KUKA KRL program: f1_Kuka_APT206T03S06.SRC

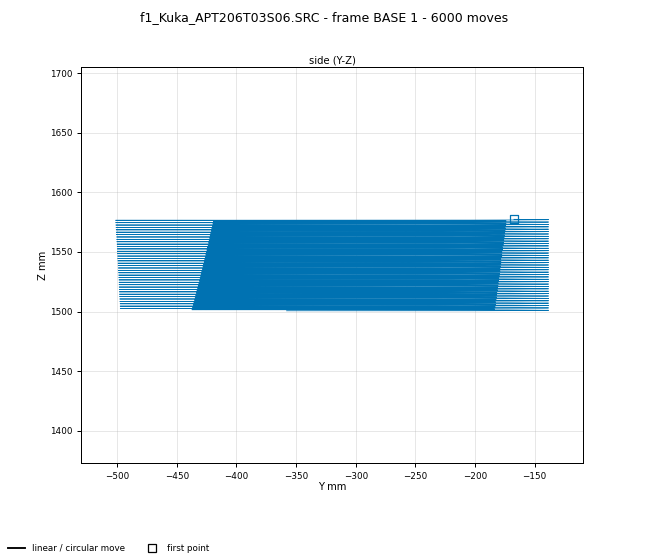
[picture p0: tool path of f1_Kuka_APT206T03S06.SRC in frame BASE 1, 6000 of 6001 moves have a stored position in this frame; points joined in program order, loops and branches not executed]
&ACCESS RVP
&REL 2
&PARAM TEMPLATE = C:\KRC\Roboter\Template\vorgabe
&PARAM EDITMASK = *
DEF f1_Kuka_APT206T03S06()


;FOLD INI;%{PE}%V3.2.0,%MKUKATPBASIS,%CINIT,%VCOMMON,%P
  ;FOLD BAS INI;%{E}%V3.2.0,%MKUKATPBASIS,%CINIT,%VINIT,%P
    GLOBAL INTERRUPT DECL 3 WHEN $STOPMESS==TRUE DO IR_STOPM ( )
    INTERRUPT ON 3
    BAS (#INITMOV,0 )
  ;ENDFOLD (BAS INI)
  ;FOLD USER INI;%{E}%V3.2.0,%MKUKATPUSER,%CINIT,%VINIT,%P
    ;Make your modifications here
  ;ENDFOLD (USER INI)
;ENDFOLD (INI)


;*** Make Null PTP Move
  PTP $pos_act

;*** Auto Load The Correct TOOL Data
  $tool=tool_data[3]

;*** Auto Load The Correct BASE Data
  $base=base_data[1]

  $ADVANCE = 5

;*** Restate Last Velocity
MMPM(30000.0)
SetRPM(6000)
LIN {X 0.095,Y -167.291,Z 1577.353,A 0.000,B 0.000,C 90.000,E1 243.512} C_DIS
LIN {X 0.027,Y -166.668,Z 1577.348,A 0.000,B 0.000,C 90.000,E1 242.666} C_DIS
LIN {X -0.056,Y -162.651,Z 1577.324,A 0.000,B 0.000,C 90.000,E1 238.329} C_DIS
LIN {X 0.006,Y -161.340,Z 1577.314,A 0.000,B 0.000,C 90.000,E1 236.548} C_DIS
LIN {X 0.048,Y -157.334,Z 1577.290,A 0.000,B 0.000,C 90.000,E1 232.110} C_DIS
LIN {X -0.019,Y -155.318,Z 1577.275,A 0.000,B 0.000,C 90.000,E1 229.461} C_DIS
LIN {X 0.019,Y -151.672,Z 1577.250,A 0.000,B 0.000,C 90.000,E1 224.960} C_DIS
LIN {X -0.040,Y -150.538,Z 1577.240,A 0.000,B 0.000,C 90.000,E1 223.176} C_DIS
LIN {X -0.007,Y -147.263,Z 1577.215,A 0.000,B 0.000,C 90.000,E1 218.624} C_DIS
LIN {X 0.050,Y -145.289,Z 1577.194,A 0.000,B 0.000,C 90.000,E1 214.945} C_DIS
LIN {X -0.041,Y -142.389,Z 1577.164,A 0.000,B 0.000,C 90.000,E1 209.461} C_DIS
LIN {X 0.005,Y -141.367,Z 1577.148,A 0.000,B 0.000,C 90.000,E1 206.668} C_DIS
LIN {X -0.017,Y -139.344,Z 1577.112,A 0.000,B 0.000,C 90.000,E1 200.174} C_DIS
LIN {X -0.011,Y -139.015,Z 1577.102,A 0.000,B 0.000,C 90.000,E1 198.308} C_DIS
LIN {X -0.015,Y -138.342,Z 1577.055,A 0.000,B 0.000,C 90.000,E1 189.905} C_DIS
LIN {X 0.004,Y -139.395,Z 1577.008,A 0.000,B 0.000,C 90.000,E1 181.489} C_DIS
LIN {X 0.058,Y -141.296,Z 1576.972,A 0.000,B 0.000,C 90.000,E1 174.951} C_DIS
LIN {X 0.016,Y -142.659,Z 1576.957,A 0.000,B 0.000,C 90.000,E1 172.186} C_DIS
LIN {X -0.034,Y -145.001,Z 1576.931,A 0.000,B 0.000,C 90.000,E1 167.589} C_DIS
LIN {X -0.045,Y -147.628,Z 1576.911,A 0.000,B 0.000,C 90.000,E1 163.921} C_DIS
LIN {X 0.033,Y -150.257,Z 1576.890,A 0.000,B 0.000,C 90.000,E1 160.242} C_DIS
LIN {X 0.047,Y -153.653,Z 1576.870,A 0.000,B 0.000,C 90.000,E1 156.613} C_DIS
LIN {X -0.036,Y -157.069,Z 1576.850,A 0.000,B 0.000,C 90.000,E1 153.050} C_DIS
LIN {X 0.042,Y -161.201,Z 1576.830,A 0.000,B 0.000,C 90.000,E1 149.459} C_DIS
LIN {X -0.009,Y -163.293,Z 1576.821,A 0.000,B 0.000,C 90.000,E1 147.709} C_DIS
LIN {X 0.001,Y -167.738,Z 1576.801,A 0.000,B 0.000,C 90.000,E1 144.196} C_DIS
LIN {X -0.087,Y -171.556,Z 1576.787,A 0.000,B 0.000,C 90.000,E1 141.618} C_DIS
LIN {X -0.046,Y -176.501,Z 1576.767,A 0.000,B 0.000,C 90.000,E1 138.162} C_DIS
LIN {X 0.080,Y -180.798,Z 1576.753,A 0.000,B 0.000,C 90.000,E1 135.567} C_DIS
LIN {X 0.065,Y -186.206,Z 1576.735,A 0.000,B 0.000,C 90.000,E1 132.204} C_DIS
LIN {X 0.004,Y -190.844,Z 1576.721,A 0.000,B 0.000,C 90.000,E1 129.725} C_DIS
LIN {X 0.038,Y -196.604,Z 1576.702,A 0.000,B 0.000,C 90.000,E1 126.423} C_DIS
LIN {X 0.006,Y -201.369,Z 1576.689,A 0.000,B 0.000,C 90.000,E1 123.992} C_DIS
LIN {X 0.013,Y -204.164,Z 1576.680,A 0.000,B 0.000,C 90.000,E1 122.418} C_DIS
LIN {X -0.014,Y -320.855,Z 1576.680,A 0.000,B 0.000,C 90.000,E1 122.418} C_DIS
LIN {X -0.039,Y -323.066,Z 1576.680,A 0.000,B 0.000,C 90.000,E1 122.388} C_DIS
LIN {X 0.035,Y -325.993,Z 1576.679,A 0.000,B 0.000,C 90.000,E1 122.260} C_DIS
LIN {X 0.100,Y -329.452,Z 1576.678,A 0.000,B 0.000,C 90.000,E1 122.005} C_DIS
LIN {X 0.070,Y -333.103,Z 1576.676,A 0.000,B 0.000,C 90.000,E1 121.592} C_DIS
LIN {X -0.223,Y -334.975,Z 1576.674,A 0.000,B 0.000,C 90.000,E1 121.337} C_DIS
LIN {X -0.056,Y -336.437,Z 1576.672,A 0.000,B 0.000,C 90.000,E1 121.003} C_DIS
LIN {X 0.068,Y -349.361,Z 1576.655,A 0.000,B 0.000,C 90.000,E1 117.897} C_DIS
LIN {X -0.105,Y -362.479,Z 1576.640,A 0.000,B 0.000,C 90.000,E1 115.207} C_DIS
LIN {X 0.113,Y -377.146,Z 1576.625,A 0.000,B 0.000,C 90.000,E1 112.514} C_DIS
LIN {X -0.183,Y -391.580,Z 1576.612,A 0.000,B 0.000,C 90.000,E1 110.248} C_DIS
LIN {X 0.123,Y -407.435,Z 1576.600,A 0.000,B 0.000,C 90.000,E1 107.946} C_DIS
LIN {X -0.208,Y -424.819,Z 1576.588,A 0.000,B 0.000,C 90.000,E1 105.788} C_DIS
LIN {X 0.185,Y -443.846,Z 1576.576,A 0.000,B 0.000,C 90.000,E1 103.592} C_DIS
LIN {X 0.113,Y -463.869,Z 1576.564,A 0.000,B 0.000,C 90.000,E1 101.591} C_DIS
LIN {X -0.162,Y -487.025,Z 1576.553,A 0.000,B 0.000,C 90.000,E1 99.557} C_DIS
LIN {X -0.235,Y -494.749,Z 1576.549,A 0.000,B 0.000,C 90.000,E1 98.916} C_DIS
LIN {X -0.117,Y -496.703,Z 1576.548,A 0.000,B 0.000,C 90.000,E1 98.681} C_DIS
LIN {X -0.073,Y -498.197,Z 1576.547,A 0.000,B 0.000,C 90.000,E1 98.454} C_DIS
LIN {X -0.153,Y -499.446,Z 1576.546,A 0.000,B 0.000,C 90.000,E1 98.219} C_DIS
LIN {X 0.192,Y -500.355,Z 1576.544,A 0.000,B 0.000,C 90.000,E1 97.936} C_DIS
LIN {X 0.043,Y -501.319,Z 1576.542,A 0.000,B 0.000,C 90.000,E1 97.466} C_DIS
LIN {X -0.168,Y -501.267,Z 1576.539,A 0.000,B 0.000,C 90.000,E1 97.004} C_DIS
LIN {X 0.122,Y -500.195,Z 1576.536,A 0.000,B 0.000,C 90.000,E1 96.486} C_DIS
LIN {X -0.009,Y -499.226,Z 1576.535,A 0.000,B 0.000,C 90.000,E1 96.258} C_DIS
LIN {X -0.137,Y -497.907,Z 1576.533,A 0.000,B 0.000,C 90.000,E1 96.030} C_DIS
LIN {X 0.044,Y -481.661,Z 1576.520,A 0.000,B 0.000,C 90.000,E1 93.555} C_DIS
LIN {X -0.017,Y -471.774,Z 1576.511,A 0.000,B 0.000,C 90.000,E1 92.064} C_DIS
LIN {X -0.040,Y -463.226,Z 1576.504,A 0.000,B 0.000,C 90.000,E1 90.802} C_DIS
LIN {X -0.187,Y -454.292,Z 1576.497,A 0.000,B 0.000,C 90.000,E1 89.542} C_DIS
LIN {X -0.018,Y -444.960,Z 1576.490,A 0.000,B 0.000,C 90.000,E1 88.224} C_DIS
LIN {X 0.026,Y -435.162,Z 1576.483,A 0.000,B 0.000,C 90.000,E1 86.906} C_DIS
LIN {X -0.192,Y -421.167,Z 1576.472,A 0.000,B 0.000,C 90.000,E1 85.065} C_DIS
LIN {X 0.006,Y -401.901,Z 1576.457,A 0.000,B 0.000,C 90.000,E1 82.299} C_DIS
LIN {X 0.185,Y -383.905,Z 1576.442,A 0.000,B 0.000,C 90.000,E1 79.454} C_DIS
LIN {X -0.013,Y -368.716,Z 1576.427,A 0.000,B 0.000,C 90.000,E1 76.881} C_DIS
LIN {X -0.045,Y -355.690,Z 1576.414,A 0.000,B 0.000,C 90.000,E1 74.519} C_DIS
LIN {X -0.198,Y -342.958,Z 1576.401,A 0.000,B 0.000,C 90.000,E1 72.127} C_DIS
LIN {X -0.144,Y -329.138,Z 1576.385,A 0.000,B 0.000,C 90.000,E1 69.337} C_DIS
LIN {X -0.054,Y -317.496,Z 1576.371,A 0.000,B 0.000,C 90.000,E1 66.794} C_DIS
LIN {X 0.006,Y -306.059,Z 1576.357,A 0.000,B 0.000,C 90.000,E1 64.204} C_DIS
LIN {X 0.045,Y -296.354,Z 1576.344,A 0.000,B 0.000,C 90.000,E1 61.897} C_DIS
LIN {X 0.140,Y -286.545,Z 1576.331,A 0.000,B 0.000,C 90.000,E1 59.537} C_DIS
LIN {X 0.017,Y -275.221,Z 1576.316,A 0.000,B 0.000,C 90.000,E1 56.834} C_DIS
LIN {X -0.067,Y -266.836,Z 1576.304,A 0.000,B 0.000,C 90.000,E1 54.769} C_DIS
LIN {X 0.128,Y -254.472,Z 1576.286,A 0.000,B 0.000,C 90.000,E1 51.537} C_DIS
LIN {X -0.100,Y -242.916,Z 1576.268,A 0.000,B 0.000,C 90.000,E1 48.324} C_DIS
LIN {X 0.003,Y -232.326,Z 1576.250,A 0.000,B 0.000,C 90.000,E1 44.960} C_DIS
LIN {X 0.061,Y -223.742,Z 1576.233,A 0.000,B 0.000,C 90.000,E1 41.919} C_DIS
LIN {X 0.110,Y -215.941,Z 1576.216,A 0.000,B 0.000,C 90.000,E1 38.830} C_DIS
LIN {X 0.031,Y -208.847,Z 1576.198,A 0.000,B 0.000,C 90.000,E1 35.724} C_DIS
LIN {X 0.045,Y -202.542,Z 1576.181,A 0.000,B 0.000,C 90.000,E1 32.546} C_DIS
LIN {X 0.031,Y -197.052,Z 1576.163,A 0.000,B 0.000,C 90.000,E1 29.333} C_DIS
LIN {X -0.059,Y -192.330,Z 1576.145,A 0.000,B 0.000,C 90.000,E1 26.104} C_DIS
LIN {X -0.007,Y -187.330,Z 1576.122,A 0.000,B 0.000,C 90.000,E1 21.972} C_DIS
LIN {X -0.033,Y -183.183,Z 1576.099,A 0.000,B 0.000,C 90.000,E1 17.819} C_DIS
LIN {X 0.054,Y -179.813,Z 1576.076,A 0.000,B 0.000,C 90.000,E1 13.592} C_DIS
LIN {X -0.068,Y -176.374,Z 1576.043,A 0.000,B 0.000,C 90.000,E1 7.701} C_DIS
LIN {X -0.029,Y -173.971,Z 1576.005,A 0.000,B 0.000,C 90.000,E1 0.859} C_DIS
LIN {X 0.097,Y -175.150,Z 1575.940,A 0.000,B 0.000,C 90.000,E1 349.218} C_DIS
LIN {X -0.078,Y -177.819,Z 1575.912,A 0.000,B 0.000,C 90.000,E1 344.157} C_DIS
LIN {X 0.041,Y -181.126,Z 1575.888,A 0.000,B 0.000,C 90.000,E1 339.880} C_DIS
LIN {X 0.075,Y -185.579,Z 1575.865,A 0.000,B 0.000,C 90.000,E1 335.665} C_DIS
LIN {X -0.008,Y -189.856,Z 1575.846,A 0.000,B 0.000,C 90.000,E1 332.359} C_DIS
LIN {X -0.062,Y -194.857,Z 1575.828,A 0.000,B 0.000,C 90.000,E1 329.076} C_DIS
LIN {X -0.022,Y -200.563,Z 1575.810,A 0.000,B 0.000,C 90.000,E1 325.801} C_DIS
LIN {X 0.064,Y -207.089,Z 1575.792,A 0.000,B 0.000,C 90.000,E1 322.557} C_DIS
LIN {X 0.077,Y -214.524,Z 1575.774,A 0.000,B 0.000,C 90.000,E1 319.380} C_DIS
LIN {X 0.023,Y -223.764,Z 1575.755,A 0.000,B 0.000,C 90.000,E1 315.891} C_DIS
LIN {X -0.040,Y -232.902,Z 1575.738,A 0.000,B 0.000,C 90.000,E1 312.852} C_DIS
LIN {X 0.002,Y -241.786,Z 1575.723,A 0.000,B 0.000,C 90.000,E1 310.216} C_DIS
LIN {X -0.050,Y -247.598,Z 1575.715,A 0.000,B 0.000,C 90.000,E1 308.749} C_DIS
LIN {X -0.028,Y -254.145,Z 1575.707,A 0.000,B 0.000,C 90.000,E1 307.282} C_DIS
LIN {X -0.028,Y -267.375,Z 1575.693,A 0.000,B 0.000,C 90.000,E1 304.771} C_DIS
LIN {X -0.044,Y -280.267,Z 1575.682,A 0.000,B 0.000,C 90.000,E1 302.673} C_DIS
LIN {X 0.109,Y -299.411,Z 1575.666,A 0.000,B 0.000,C 90.000,E1 299.922} C_DIS
LIN {X 0.048,Y -311.876,Z 1575.657,A 0.000,B 0.000,C 90.000,E1 298.281} C_DIS
LIN {X -0.027,Y -326.927,Z 1575.646,A 0.000,B 0.000,C 90.000,E1 296.360} C_DIS
LIN {X 0.062,Y -339.369,Z 1575.638,A 0.000,B 0.000,C 90.000,E1 294.771} C_DIS
LIN {X -0.090,Y -361.712,Z 1575.623,A 0.000,B 0.000,C 90.000,E1 292.078} C_DIS
LIN {X 0.149,Y -374.611,Z 1575.614,A 0.000,B 0.000,C 90.000,E1 290.556} C_DIS
LIN {X 0.113,Y -384.575,Z 1575.608,A 0.000,B 0.000,C 90.000,E1 289.396} C_DIS
LIN {X 0.036,Y -391.545,Z 1575.603,A 0.000,B 0.000,C 90.000,E1 288.544} C_DIS
LIN {X 0.079,Y -399.857,Z 1575.597,A 0.000,B 0.000,C 90.000,E1 287.402} C_DIS
LIN {X -0.055,Y -403.577,Z 1575.594,A 0.000,B 0.000,C 90.000,E1 286.858} C_DIS
LIN {X -0.075,Y -408.391,Z 1575.589,A 0.000,B 0.000,C 90.000,E1 286.024} C_DIS
LIN {X -0.160,Y -411.130,Z 1575.586,A 0.000,B 0.000,C 90.000,E1 285.481} C_DIS
LIN {X 0.060,Y -413.511,Z 1575.583,A 0.000,B 0.000,C 90.000,E1 284.898} C_DIS
LIN {X 0.129,Y -416.344,Z 1575.578,A 0.000,B 0.000,C 90.000,E1 284.064} C_DIS
LIN {X -0.018,Y -417.781,Z 1575.575,A 0.000,B 0.000,C 90.000,E1 283.536} C_DIS
LIN {X -0.153,Y -418.766,Z 1575.572,A 0.000,B 0.000,C 90.000,E1 283.008} C_DIS
LIN {X 0.220,Y -419.304,Z 1575.569,A 0.000,B 0.000,C 90.000,E1 282.411} C_DIS
LIN {X 0.097,Y -419.380,Z 1575.566,A 0.000,B 0.000,C 90.000,E1 281.883} C_DIS
LIN {X -0.107,Y -418.925,Z 1575.563,A 0.000,B 0.000,C 90.000,E1 281.366} C_DIS
LIN {X -0.225,Y -417.916,Z 1575.560,A 0.000,B 0.000,C 90.000,E1 280.838} C_DIS
LIN {X 0.063,Y -416.325,Z 1575.557,A 0.000,B 0.000,C 90.000,E1 280.254} C_DIS
LIN {X -0.067,Y -414.093,Z 1575.554,A 0.000,B 0.000,C 90.000,E1 279.726} C_DIS
LIN {X -0.005,Y -412.764,Z 1575.552,A 0.000,B 0.000,C 90.000,E1 279.443} C_DIS
LIN {X -0.157,Y -409.484,Z 1575.549,A 0.000,B 0.000,C 90.000,E1 278.916} C_DIS
LIN {X 0.014,Y -405.457,Z 1575.546,A 0.000,B 0.000,C 90.000,E1 278.341} C_DIS
LIN {X -0.179,Y -400.748,Z 1575.543,A 0.000,B 0.000,C 90.000,E1 277.814} C_DIS
LIN {X 0.036,Y -395.299,Z 1575.540,A 0.000,B 0.000,C 90.000,E1 277.239} C_DIS
LIN {X 0.065,Y -389.417,Z 1575.537,A 0.000,B 0.000,C 90.000,E1 276.720} C_DIS
LIN {X -0.010,Y -383.356,Z 1575.535,A 0.000,B 0.000,C 90.000,E1 276.258} C_DIS
LIN {X -0.011,Y -373.859,Z 1575.531,A 0.000,B 0.000,C 90.000,E1 275.625} C_DIS
LIN {X -0.175,Y -364.295,Z 1575.528,A 0.000,B 0.000,C 90.000,E1 275.106} C_DIS
LIN {X 0.037,Y -354.579,Z 1575.526,A 0.000,B 0.000,C 90.000,E1 274.588} C_DIS
LIN {X -0.165,Y -345.037,Z 1575.523,A 0.000,B 0.000,C 90.000,E1 274.188} C_DIS
LIN {X 0.165,Y -335.255,Z 1575.521,A 0.000,B 0.000,C 90.000,E1 273.726} C_DIS
LIN {X -0.025,Y -322.280,Z 1575.518,A 0.000,B 0.000,C 90.000,E1 273.269} C_DIS
LIN {X 0.106,Y -312.075,Z 1575.516,A 0.000,B 0.000,C 90.000,E1 272.922} C_DIS
LIN {X 0.125,Y -301.579,Z 1575.515,A 0.000,B 0.000,C 90.000,E1 272.636} C_DIS
LIN {X 0.116,Y -290.375,Z 1575.514,A 0.000,B 0.000,C 90.000,E1 272.407} C_DIS
LIN {X 0.057,Y -277.059,Z 1575.512,A 0.000,B 0.000,C 90.000,E1 272.236} C_DIS
LIN {X -0.089,Y -257.665,Z 1575.511,A 0.000,B 0.000,C 90.000,E1 272.064} C_DIS
LIN {X 0.109,Y -244.909,Z 1575.511,A 0.000,B 0.000,C 90.000,E1 271.949} C_DIS
LIN {X 0.058,Y -238.715,Z 1575.511,A 0.000,B 0.000,C 90.000,E1 271.949} C_DIS
LIN {X 0.026,Y -181.269,Z 1575.511,A 0.000,B 0.000,C 90.000,E1 271.949} C_DIS
LIN {X -0.068,Y -181.572,Z 1575.502,A 0.000,B 0.000,C 90.000,E1 270.458} C_DIS
LIN {X 0.015,Y -180.953,Z 1575.481,A 0.000,B 0.000,C 90.000,E1 266.560} C_DIS
LIN {X -0.048,Y -180.830,Z 1575.472,A 0.000,B 0.000,C 90.000,E1 264.894} C_DIS
LIN {X 0.032,Y -178.936,Z 1575.443,A 0.000,B 0.000,C 90.000,E1 259.803} C_DIS
LIN {X -0.100,Y -175.984,Z 1575.415,A 0.000,B 0.000,C 90.000,E1 254.755} C_DIS
LIN {X 0.015,Y -175.481,Z 1575.410,A 0.000,B 0.000,C 90.000,E1 253.866} C_DIS
LIN {X 0.072,Y -172.227,Z 1575.387,A 0.000,B 0.000,C 90.000,E1 249.571} C_DIS
LIN {X 0.049,Y -171.704,Z 1575.382,A 0.000,B 0.000,C 90.000,E1 248.720} C_DIS
LIN {X -0.026,Y -167.298,Z 1575.353,A 0.000,B 0.000,C 90.000,E1 243.563} C_DIS
LIN {X 0.056,Y -166.676,Z 1575.348,A 0.000,B 0.000,C 90.000,E1 242.666} C_DIS
LIN {X -0.029,Y -162.658,Z 1575.324,A 0.000,B 0.000,C 90.000,E1 238.329} C_DIS
LIN {X 0.033,Y -161.347,Z 1575.314,A 0.000,B 0.000,C 90.000,E1 236.548} C_DIS
LIN {X 0.075,Y -157.342,Z 1575.290,A 0.000,B 0.000,C 90.000,E1 232.110} C_DIS
LIN {X 0.008,Y -155.327,Z 1575.275,A 0.000,B 0.000,C 90.000,E1 229.461} C_DIS
LIN {X -0.062,Y -151.679,Z 1575.250,A 0.000,B 0.000,C 90.000,E1 225.000} C_DIS
LIN {X -0.014,Y -150.543,Z 1575.240,A 0.000,B 0.000,C 90.000,E1 223.176} C_DIS
LIN {X 0.020,Y -147.269,Z 1575.215,A 0.000,B 0.000,C 90.000,E1 218.624} C_DIS
LIN {X -0.008,Y -145.296,Z 1575.194,A 0.000,B 0.000,C 90.000,E1 214.978} C_DIS
LIN {X -0.015,Y -142.392,Z 1575.164,A 0.000,B 0.000,C 90.000,E1 209.461} C_DIS
LIN {X 0.031,Y -141.372,Z 1575.148,A 0.000,B 0.000,C 90.000,E1 206.668} C_DIS
LIN {X 0.009,Y -139.346,Z 1575.112,A 0.000,B 0.000,C 90.000,E1 200.174} C_DIS
LIN {X 0.014,Y -139.018,Z 1575.102,A 0.000,B 0.000,C 90.000,E1 198.308} C_DIS
LIN {X 0.010,Y -138.343,Z 1575.055,A 0.000,B 0.000,C 90.000,E1 189.905} C_DIS
LIN {X 0.029,Y -139.392,Z 1575.008,A 0.000,B 0.000,C 90.000,E1 181.489} C_DIS
LIN {X -0.057,Y -141.291,Z 1574.972,A 0.000,B 0.000,C 90.000,E1 175.008} C_DIS
LIN {X 0.042,Y -142.654,Z 1574.957,A 0.000,B 0.000,C 90.000,E1 172.186} C_DIS
LIN {X -0.008,Y -144.994,Z 1574.931,A 0.000,B 0.000,C 90.000,E1 167.589} C_DIS
LIN {X -0.019,Y -147.621,Z 1574.911,A 0.000,B 0.000,C 90.000,E1 163.921} C_DIS
LIN {X 0.059,Y -150.248,Z 1574.890,A 0.000,B 0.000,C 90.000,E1 160.242} C_DIS
LIN {X -0.067,Y -153.643,Z 1574.870,A 0.000,B 0.000,C 90.000,E1 156.666} C_DIS
LIN {X -0.009,Y -157.059,Z 1574.850,A 0.000,B 0.000,C 90.000,E1 153.050} C_DIS
LIN {X 0.071,Y -161.189,Z 1574.830,A 0.000,B 0.000,C 90.000,E1 149.459} C_DIS
LIN {X 0.019,Y -163.281,Z 1574.821,A 0.000,B 0.000,C 90.000,E1 147.709} C_DIS
LIN {X 0.029,Y -167.725,Z 1574.801,A 0.000,B 0.000,C 90.000,E1 144.196} C_DIS
LIN {X -0.058,Y -171.543,Z 1574.787,A 0.000,B 0.000,C 90.000,E1 141.618} C_DIS
LIN {X -0.016,Y -176.486,Z 1574.768,A 0.000,B 0.000,C 90.000,E1 138.162} C_DIS
LIN {X 0.109,Y -180.783,Z 1574.753,A 0.000,B 0.000,C 90.000,E1 135.567} C_DIS
LIN {X -0.030,Y -186.190,Z 1574.735,A 0.000,B 0.000,C 90.000,E1 132.243} C_DIS
LIN {X 0.035,Y -190.827,Z 1574.721,A 0.000,B 0.000,C 90.000,E1 129.725} C_DIS
LIN {X -0.047,Y -196.587,Z 1574.703,A 0.000,B 0.000,C 90.000,E1 126.457} C_DIS
LIN {X 0.037,Y -201.354,Z 1574.689,A 0.000,B 0.000,C 90.000,E1 123.992} C_DIS
LIN {X -0.027,Y -204.096,Z 1574.680,A 0.000,B 0.000,C 90.000,E1 122.467} C_DIS
LIN {X -0.078,Y -320.847,Z 1574.680,A 0.000,B 0.000,C 90.000,E1 122.467} C_DIS
LIN {X -0.162,Y -323.865,Z 1574.680,A 0.000,B 0.000,C 90.000,E1 122.418} C_DIS
LIN {X -0.054,Y -326.764,Z 1574.679,A 0.000,B 0.000,C 90.000,E1 122.260} C_DIS
LIN {X -0.011,Y -330.385,Z 1574.677,A 0.000,B 0.000,C 90.000,E1 121.957} C_DIS
LIN {X 0.095,Y -333.985,Z 1574.675,A 0.000,B 0.000,C 90.000,E1 121.465} C_DIS
LIN {X -0.073,Y -335.662,Z 1574.673,A 0.000,B 0.000,C 90.000,E1 121.180} C_DIS
LIN {X 0.015,Y -349.958,Z 1574.654,A 0.000,B 0.000,C 90.000,E1 117.769} C_DIS
LIN {X -0.143,Y -363.150,Z 1574.639,A 0.000,B 0.000,C 90.000,E1 115.079} C_DIS
LIN {X 0.092,Y -377.897,Z 1574.624,A 0.000,B 0.000,C 90.000,E1 112.386} C_DIS
LIN {X -0.189,Y -392.407,Z 1574.612,A 0.000,B 0.000,C 90.000,E1 110.120} C_DIS
LIN {X 0.133,Y -408.345,Z 1574.599,A 0.000,B 0.000,C 90.000,E1 107.819} C_DIS
LIN {X -0.181,Y -425.818,Z 1574.587,A 0.000,B 0.000,C 90.000,E1 105.662} C_DIS
LIN {X 0.139,Y -444.926,Z 1574.575,A 0.000,B 0.000,C 90.000,E1 103.480} C_DIS
LIN {X 0.149,Y -464.980,Z 1574.564,A 0.000,B 0.000,C 90.000,E1 101.478} C_DIS
LIN {X -0.038,Y -488.170,Z 1574.552,A 0.000,B 0.000,C 90.000,E1 99.443} C_DIS
LIN {X -0.190,Y -493.404,Z 1574.550,A 0.000,B 0.000,C 90.000,E1 99.029} C_DIS
LIN {X -0.082,Y -495.600,Z 1574.549,A 0.000,B 0.000,C 90.000,E1 98.803} C_DIS
LIN {X -0.110,Y -497.434,Z 1574.547,A 0.000,B 0.000,C 90.000,E1 98.568} C_DIS
LIN {X -0.213,Y -498.815,Z 1574.546,A 0.000,B 0.000,C 90.000,E1 98.341} C_DIS
LIN {X 0.126,Y -500.604,Z 1574.543,A 0.000,B 0.000,C 90.000,E1 97.814} C_DIS
LIN {X -0.095,Y -501.274,Z 1574.541,A 0.000,B 0.000,C 90.000,E1 97.352} C_DIS
LIN {X 0.193,Y -500.943,Z 1574.538,A 0.000,B 0.000,C 90.000,E1 96.834} C_DIS
LIN {X -0.012,Y -499.559,Z 1574.535,A 0.000,B 0.000,C 90.000,E1 96.372} C_DIS
LIN {X -0.142,Y -498.401,Z 1574.534,A 0.000,B 0.000,C 90.000,E1 96.144} C_DIS
LIN {X -0.151,Y -485.465,Z 1574.523,A 0.000,B 0.000,C 90.000,E1 94.188} C_DIS
LIN {X -0.118,Y -475.726,Z 1574.515,A 0.000,B 0.000,C 90.000,E1 92.694} C_DIS
LIN {X 0.187,Y -465.673,Z 1574.506,A 0.000,B 0.000,C 90.000,E1 91.146} C_DIS
LIN {X 0.069,Y -456.832,Z 1574.499,A 0.000,B 0.000,C 90.000,E1 89.885} C_DIS
LIN {X -0.175,Y -447.619,Z 1574.492,A 0.000,B 0.000,C 90.000,E1 88.625} C_DIS
LIN {X -0.087,Y -437.962,Z 1574.485,A 0.000,B 0.000,C 90.000,E1 87.306} C_DIS
LIN {X 0.022,Y -425.988,Z 1574.476,A 0.000,B 0.000,C 90.000,E1 85.698} C_DIS
LIN {X -0.168,Y -408.379,Z 1574.463,A 0.000,B 0.000,C 90.000,E1 83.280} C_DIS
LIN {X 0.151,Y -389.972,Z 1574.447,A 0.000,B 0.000,C 90.000,E1 80.443} C_DIS
LIN {X 0.128,Y -369.444,Z 1574.428,A 0.000,B 0.000,C 90.000,E1 76.992} C_DIS
LIN {X 0.115,Y -356.384,Z 1574.415,A 0.000,B 0.000,C 90.000,E1 74.629} C_DIS
LIN {X -0.034,Y -345.224,Z 1574.403,A 0.000,B 0.000,C 90.000,E1 72.543} C_DIS
LIN {X 0.060,Y -329.742,Z 1574.386,A 0.000,B 0.000,C 90.000,E1 69.444} C_DIS
LIN {X -0.018,Y -316.635,Z 1574.370,A 0.000,B 0.000,C 90.000,E1 66.613} C_DIS
LIN {X 0.015,Y -305.186,Z 1574.356,A 0.000,B 0.000,C 90.000,E1 64.024} C_DIS
LIN {X 0.030,Y -295.451,Z 1574.343,A 0.000,B 0.000,C 90.000,E1 61.719} C_DIS
LIN {X -0.149,Y -285.589,Z 1574.330,A 0.000,B 0.000,C 90.000,E1 59.410} C_DIS
LIN {X 0.095,Y -274.341,Z 1574.315,A 0.000,B 0.000,C 90.000,E1 56.628} C_DIS
LIN {X -0.007,Y -266.015,Z 1574.303,A 0.000,B 0.000,C 90.000,E1 54.562} C_DIS
LIN {X -0.039,Y -253.733,Z 1574.285,A 0.000,B 0.000,C 90.000,E1 51.376} C_DIS
LIN {X 0.067,Y -242.256,Z 1574.267,A 0.000,B 0.000,C 90.000,E1 48.081} C_DIS
LIN {X -0.017,Y -231.760,Z 1574.249,A 0.000,B 0.000,C 90.000,E1 44.757} C_DIS
LIN {X -0.130,Y -223.234,Z 1574.232,A 0.000,B 0.000,C 90.000,E1 41.757} C_DIS
LIN {X 0.078,Y -215.496,Z 1574.215,A 0.000,B 0.000,C 90.000,E1 38.624} C_DIS
LIN {X -0.009,Y -208.484,Z 1574.197,A 0.000,B 0.000,C 90.000,E1 35.518} C_DIS
LIN {X -0.001,Y -202.268,Z 1574.180,A 0.000,B 0.000,C 90.000,E1 32.339} C_DIS
LIN {X -0.023,Y -196.843,Z 1574.162,A 0.000,B 0.000,C 90.000,E1 29.127} C_DIS
LIN {X 0.052,Y -192.183,Z 1574.144,A 0.000,B 0.000,C 90.000,E1 25.848} C_DIS
LIN {X 0.095,Y -187.263,Z 1574.121,A 0.000,B 0.000,C 90.000,E1 21.716} C_DIS
LIN {X 0.001,Y -183.167,Z 1574.098,A 0.000,B 0.000,C 90.000,E1 17.583} C_DIS
LIN {X 0.016,Y -179.309,Z 1574.070,A 0.000,B 0.000,C 90.000,E1 12.535} C_DIS
LIN {X -0.007,Y -176.097,Z 1574.037,A 0.000,B 0.000,C 90.000,E1 6.606} C_DIS
LIN {X -0.032,Y -174.013,Z 1573.997,A 0.000,B 0.000,C 90.000,E1 359.542} C_DIS
LIN {X -0.057,Y -175.411,Z 1573.940,A 0.000,B 0.000,C 90.000,E1 349.275} C_DIS
LIN {X -0.050,Y -178.082,Z 1573.912,A 0.000,B 0.000,C 90.000,E1 344.157} C_DIS
LIN {X 0.078,Y -181.397,Z 1573.888,A 0.000,B 0.000,C 90.000,E1 339.880} C_DIS
LIN {X -0.048,Y -185.808,Z 1573.865,A 0.000,B 0.000,C 90.000,E1 335.717} C_DIS
LIN {X 0.045,Y -190.072,Z 1573.847,A 0.000,B 0.000,C 90.000,E1 332.359} C_DIS
LIN {X -0.003,Y -195.024,Z 1573.828,A 0.000,B 0.000,C 90.000,E1 329.076} C_DIS
LIN {X 0.044,Y -200.698,Z 1573.810,A 0.000,B 0.000,C 90.000,E1 325.801} C_DIS
LIN {X -0.030,Y -207.204,Z 1573.792,A 0.000,B 0.000,C 90.000,E1 322.603} C_DIS
LIN {X -0.149,Y -214.589,Z 1573.775,A 0.000,B 0.000,C 90.000,E1 319.461} C_DIS
LIN {X 0.105,Y -223.812,Z 1573.755,A 0.000,B 0.000,C 90.000,E1 315.891} C_DIS
LIN {X 0.046,Y -232.891,Z 1573.738,A 0.000,B 0.000,C 90.000,E1 312.852} C_DIS
LIN {X -0.066,Y -241.728,Z 1573.724,A 0.000,B 0.000,C 90.000,E1 310.253} C_DIS
LIN {X 0.039,Y -247.490,Z 1573.715,A 0.000,B 0.000,C 90.000,E1 308.749} C_DIS
LIN {X 0.063,Y -254.005,Z 1573.707,A 0.000,B 0.000,C 90.000,E1 307.282} C_DIS
LIN {X -0.057,Y -265.240,Z 1573.695,A 0.000,B 0.000,C 90.000,E1 305.152} C_DIS
LIN {X 0.030,Y -275.640,Z 1573.685,A 0.000,B 0.000,C 90.000,E1 303.372} C_DIS
LIN {X -0.134,Y -289.471,Z 1573.674,A 0.000,B 0.000,C 90.000,E1 301.337} C_DIS
LIN {X 0.085,Y -306.745,Z 1573.661,A 0.000,B 0.000,C 90.000,E1 298.949} C_DIS
LIN {X 0.064,Y -321.753,Z 1573.650,A 0.000,B 0.000,C 90.000,E1 297.001} C_DIS
LIN {X -0.114,Y -336.586,Z 1573.640,A 0.000,B 0.000,C 90.000,E1 295.155} C_DIS
LIN {X -0.093,Y -353.914,Z 1573.628,A 0.000,B 0.000,C 90.000,E1 293.003} C_DIS
LIN {X -0.083,Y -369.209,Z 1573.618,A 0.000,B 0.000,C 90.000,E1 291.227} C_DIS
LIN {X 0.064,Y -381.785,Z 1573.610,A 0.000,B 0.000,C 90.000,E1 289.758} C_DIS
LIN {X 0.072,Y -388.863,Z 1573.605,A 0.000,B 0.000,C 90.000,E1 288.906} C_DIS
LIN {X 0.032,Y -395.484,Z 1573.600,A 0.000,B 0.000,C 90.000,E1 288.055} C_DIS
LIN {X -0.064,Y -401.491,Z 1573.596,A 0.000,B 0.000,C 90.000,E1 287.221} C_DIS
LIN {X -0.108,Y -406.707,Z 1573.591,A 0.000,B 0.000,C 90.000,E1 286.386} C_DIS
LIN {X -0.203,Y -409.746,Z 1573.588,A 0.000,B 0.000,C 90.000,E1 285.843} C_DIS
LIN {X -0.168,Y -413.518,Z 1573.583,A 0.000,B 0.000,C 90.000,E1 285.009} C_DIS
LIN {X -0.104,Y -416.483,Z 1573.579,A 0.000,B 0.000,C 90.000,E1 284.175} C_DIS
LIN {X 0.152,Y -417.968,Z 1573.576,A 0.000,B 0.000,C 90.000,E1 283.592} C_DIS
LIN {X 0.017,Y -419.068,Z 1573.573,A 0.000,B 0.000,C 90.000,E1 283.063} C_DIS
LIN {X -0.109,Y -419.655,Z 1573.570,A 0.000,B 0.000,C 90.000,E1 282.535} C_DIS
LIN {X 0.182,Y -419.835,Z 1573.567,A 0.000,B 0.000,C 90.000,E1 281.951} C_DIS
LIN {X 0.066,Y -419.470,Z 1573.563,A 0.000,B 0.000,C 90.000,E1 281.422} C_DIS
LIN {X -0.051,Y -418.568,Z 1573.560,A 0.000,B 0.000,C 90.000,E1 280.894} C_DIS
LIN {X -0.171,Y -417.121,Z 1573.557,A 0.000,B 0.000,C 90.000,E1 280.366} C_DIS
LIN {X 0.041,Y -415.016,Z 1573.554,A 0.000,B 0.000,C 90.000,E1 279.792} C_DIS
LIN {X -0.093,Y -412.268,Z 1573.551,A 0.000,B 0.000,C 90.000,E1 279.265} C_DIS
LIN {X 0.093,Y -408.781,Z 1573.548,A 0.000,B 0.000,C 90.000,E1 278.690} C_DIS
LIN {X -0.081,Y -404.551,Z 1573.545,A 0.000,B 0.000,C 90.000,E1 278.163} C_DIS
LIN {X 0.063,Y -399.489,Z 1573.542,A 0.000,B 0.000,C 90.000,E1 277.587} C_DIS
LIN {X -0.092,Y -393.814,Z 1573.539,A 0.000,B 0.000,C 90.000,E1 277.068} C_DIS
LIN {X 0.079,Y -387.951,Z 1573.536,A 0.000,B 0.000,C 90.000,E1 276.549} C_DIS
LIN {X 0.101,Y -381.690,Z 1573.534,A 0.000,B 0.000,C 90.000,E1 276.087} C_DIS
LIN {X 0.049,Y -375.422,Z 1573.532,A 0.000,B 0.000,C 90.000,E1 275.682} C_DIS
LIN {X -0.144,Y -369.060,Z 1573.530,A 0.000,B 0.000,C 90.000,E1 275.334} C_DIS
LIN {X -0.071,Y -359.451,Z 1573.527,A 0.000,B 0.000,C 90.000,E1 274.821} C_DIS
LIN {X -0.030,Y -349.762,Z 1573.524,A 0.000,B 0.000,C 90.000,E1 274.359} C_DIS
LIN {X -0.058,Y -340.294,Z 1573.522,A 0.000,B 0.000,C 90.000,E1 273.955} C_DIS
LIN {X 0.007,Y -327.444,Z 1573.519,A 0.000,B 0.000,C 90.000,E1 273.440} C_DIS
LIN {X -0.033,Y -320.877,Z 1573.518,A 0.000,B 0.000,C 90.000,E1 273.212} C_DIS
LIN {X 0.141,Y -310.524,Z 1573.516,A 0.000,B 0.000,C 90.000,E1 272.865} C_DIS
LIN {X -0.050,Y -300.310,Z 1573.515,A 0.000,B 0.000,C 90.000,E1 272.636} C_DIS
LIN {X 0.033,Y -292.758,Z 1573.514,A 0.000,B 0.000,C 90.000,E1 272.465} C_DIS
LIN {X -0.076,Y -279.445,Z 1573.513,A 0.000,B 0.000,C 90.000,E1 272.293} C_DIS
LIN {X 0.043,Y -261.100,Z 1573.511,A 0.000,B 0.000,C 90.000,E1 272.064} C_DIS
LIN {X -0.111,Y -245.733,Z 1573.511,A 0.000,B 0.000,C 90.000,E1 272.007} C_DIS
LIN {X 0.090,Y -240.633,Z 1573.511,A 0.000,B 0.000,C 90.000,E1 271.949} C_DIS
LIN {X 0.035,Y -181.268,Z 1573.511,A 0.000,B 0.000,C 90.000,E1 271.949} C_DIS
LIN {X -0.045,Y -181.580,Z 1573.501,A 0.000,B 0.000,C 90.000,E1 270.229} C_DIS
LIN {X -0.055,Y -180.891,Z 1573.473,A 0.000,B 0.000,C 90.000,E1 265.179} C_DIS
LIN {X 0.007,Y -179.016,Z 1573.445,A 0.000,B 0.000,C 90.000,E1 260.095} C_DIS
LIN {X 0.102,Y -178.642,Z 1573.440,A 0.000,B 0.000,C 90.000,E1 259.218} C_DIS
LIN {X -0.001,Y -175.693,Z 1573.412,A 0.000,B 0.000,C 90.000,E1 254.157} C_DIS
LIN {X 0.010,Y -172.409,Z 1573.388,A 0.000,B 0.000,C 90.000,E1 249.880} C_DIS
LIN {X 0.026,Y -171.224,Z 1573.379,A 0.000,B 0.000,C 90.000,E1 248.156} C_DIS
LIN {X 0.003,Y -167.506,Z 1573.355,A 0.000,B 0.000,C 90.000,E1 243.845} C_DIS
LIN {X -0.065,Y -166.901,Z 1573.350,A 0.000,B 0.000,C 90.000,E1 242.999} C_DIS
LIN {X -0.012,Y -162.208,Z 1573.321,A 0.000,B 0.000,C 90.000,E1 237.740} C_DIS
LIN {X 0.041,Y -160.785,Z 1573.311,A 0.000,B 0.000,C 90.000,E1 235.960} C_DIS
LIN {X 0.012,Y -157.577,Z 1573.291,A 0.000,B 0.000,C 90.000,E1 232.431} C_DIS
LIN {X 0.046,Y -155.608,Z 1573.276,A 0.000,B 0.000,C 90.000,E1 229.747} C_DIS
LIN {X -0.011,Y -151.888,Z 1573.252,A 0.000,B 0.000,C 90.000,E1 225.283} C_DIS
LIN {X 0.008,Y -150.115,Z 1573.236,A 0.000,B 0.000,C 90.000,E1 222.567} C_DIS
LIN {X 0.026,Y -146.909,Z 1573.211,A 0.000,B 0.000,C 90.000,E1 218.016} C_DIS
LIN {X -0.073,Y -145.497,Z 1573.196,A 0.000,B 0.000,C 90.000,E1 215.311} C_DIS
LIN {X 0.045,Y -142.902,Z 1573.171,A 0.000,B 0.000,C 90.000,E1 210.669} C_DIS
LIN {X -0.024,Y -141.522,Z 1573.150,A 0.000,B 0.000,C 90.000,E1 207.001} C_DIS
LIN {X 0.019,Y -139.395,Z 1573.114,A 0.000,B 0.000,C 90.000,E1 200.482} C_DIS
LIN {X 0.070,Y -139.107,Z 1573.104,A 0.000,B 0.000,C 90.000,E1 198.598} C_DIS
LIN {X 0.061,Y -138.353,Z 1573.057,A 0.000,B 0.000,C 90.000,E1 190.197} C_DIS
LIN {X 0.055,Y -139.511,Z 1573.005,A 0.000,B 0.000,C 90.000,E1 180.859} C_DIS
LIN {X -0.004,Y -141.153,Z 1572.974,A 0.000,B 0.000,C 90.000,E1 175.298} C_DIS
LIN {X -0.033,Y -142.533,Z 1572.958,A 0.000,B 0.000,C 90.000,E1 172.527} C_DIS
LIN {X 0.035,Y -144.803,Z 1572.933,A 0.000,B 0.000,C 90.000,E1 167.881} C_DIS
LIN {X 0.023,Y -147.421,Z 1572.912,A 0.000,B 0.000,C 90.000,E1 164.212} C_DIS
LIN {X 0.052,Y -149.998,Z 1572.892,A 0.000,B 0.000,C 90.000,E1 160.550} C_DIS
LIN {X 0.059,Y -153.328,Z 1572.872,A 0.000,B 0.000,C 90.000,E1 156.922} C_DIS
LIN {X -0.029,Y -155.027,Z 1572.862,A 0.000,B 0.000,C 90.000,E1 155.153} C_DIS
LIN {X -0.007,Y -158.674,Z 1572.842,A 0.000,B 0.000,C 90.000,E1 151.563} C_DIS
LIN {X 0.075,Y -161.953,Z 1572.827,A 0.000,B 0.000,C 90.000,E1 148.869} C_DIS
LIN {X -0.041,Y -166.145,Z 1572.808,A 0.000,B 0.000,C 90.000,E1 145.388} C_DIS
LIN {X -0.045,Y -171.157,Z 1572.788,A 0.000,B 0.000,C 90.000,E1 141.904} C_DIS
LIN {X -0.010,Y -176.035,Z 1572.769,A 0.000,B 0.000,C 90.000,E1 138.447} C_DIS
LIN {X -0.014,Y -180.290,Z 1572.755,A 0.000,B 0.000,C 90.000,E1 135.891} C_DIS
LIN {X -0.042,Y -185.702,Z 1572.736,A 0.000,B 0.000,C 90.000,E1 132.528} C_DIS
LIN {X 0.009,Y -190.307,Z 1572.722,A 0.000,B 0.000,C 90.000,E1 130.011} C_DIS
LIN {X 0.057,Y -197.634,Z 1572.699,A 0.000,B 0.000,C 90.000,E1 125.884} C_DIS
LIN {X -0.013,Y -200.891,Z 1572.690,A 0.000,B 0.000,C 90.000,E1 124.278} C_DIS
LIN {X 0.015,Y -204.017,Z 1572.681,A 0.000,B 0.000,C 90.000,E1 122.498} C_DIS
LIN {X -0.025,Y -320.360,Z 1572.681,A 0.000,B 0.000,C 90.000,E1 122.498} C_DIS
LIN {X 0.049,Y -321.886,Z 1572.680,A 0.000,B 0.000,C 90.000,E1 122.467} C_DIS
LIN {X -0.106,Y -326.059,Z 1572.680,A 0.000,B 0.000,C 90.000,E1 122.339} C_DIS
LIN {X 0.189,Y -328.326,Z 1572.679,A 0.000,B 0.000,C 90.000,E1 122.133} C_DIS
LIN {X -0.124,Y -331.434,Z 1572.677,A 0.000,B 0.000,C 90.000,E1 121.878} C_DIS
LIN {X -0.197,Y -335.013,Z 1572.674,A 0.000,B 0.000,C 90.000,E1 121.337} C_DIS
LIN {X 0.050,Y -337.648,Z 1572.670,A 0.000,B 0.000,C 90.000,E1 120.669} C_DIS
LIN {X 0.042,Y -349.337,Z 1572.655,A 0.000,B 0.000,C 90.000,E1 117.897} C_DIS
LIN {X -0.138,Y -362.460,Z 1572.640,A 0.000,B 0.000,C 90.000,E1 115.207} C_DIS
LIN {X 0.084,Y -377.125,Z 1572.625,A 0.000,B 0.000,C 90.000,E1 112.514} C_DIS
LIN {X -0.213,Y -391.561,Z 1572.612,A 0.000,B 0.000,C 90.000,E1 110.248} C_DIS
LIN {X 0.091,Y -407.417,Z 1572.600,A 0.000,B 0.000,C 90.000,E1 107.946} C_DIS
LIN {X -0.242,Y -424.804,Z 1572.588,A 0.000,B 0.000,C 90.000,E1 105.788} C_DIS
LIN {X 0.160,Y -443.821,Z 1572.576,A 0.000,B 0.000,C 90.000,E1 103.592} C_DIS
LIN {X 0.088,Y -463.843,Z 1572.564,A 0.000,B 0.000,C 90.000,E1 101.591} C_DIS
LIN {X -0.208,Y -487.028,Z 1572.553,A 0.000,B 0.000,C 90.000,E1 99.557} C_DIS
LIN {X 0.227,Y -494.681,Z 1572.549,A 0.000,B 0.000,C 90.000,E1 98.859} C_DIS
LIN {X -0.067,Y -496.521,Z 1572.548,A 0.000,B 0.000,C 90.000,E1 98.681} C_DIS
LIN {X -0.226,Y -498.131,Z 1572.547,A 0.000,B 0.000,C 90.000,E1 98.454} C_DIS
LIN {X 0.182,Y -499.331,Z 1572.545,A 0.000,B 0.000,C 90.000,E1 98.163} C_DIS
LIN {X -0.040,Y -500.773,Z 1572.543,A 0.000,B 0.000,C 90.000,E1 97.701} C_DIS
LIN {X 0.241,Y -501.151,Z 1572.540,A 0.000,B 0.000,C 90.000,E1 97.182} C_DIS
LIN {X 0.034,Y -500.529,Z 1572.537,A 0.000,B 0.000,C 90.000,E1 96.720} C_DIS
LIN {X -0.171,Y -498.807,Z 1572.535,A 0.000,B 0.000,C 90.000,E1 96.258} C_DIS
LIN {X 0.245,Y -497.432,Z 1572.533,A 0.000,B 0.000,C 90.000,E1 95.967} C_DIS
LIN {X -0.127,Y -481.237,Z 1572.520,A 0.000,B 0.000,C 90.000,E1 93.555} C_DIS
LIN {X -0.191,Y -471.381,Z 1572.511,A 0.000,B 0.000,C 90.000,E1 92.064} C_DIS
LIN {X -0.211,Y -462.855,Z 1572.504,A 0.000,B 0.000,C 90.000,E1 90.802} C_DIS
LIN {X 0.089,Y -453.895,Z 1572.497,A 0.000,B 0.000,C 90.000,E1 89.484} C_DIS
LIN {X -0.193,Y -444.579,Z 1572.490,A 0.000,B 0.000,C 90.000,E1 88.224} C_DIS
LIN {X -0.156,Y -434.793,Z 1572.483,A 0.000,B 0.000,C 90.000,E1 86.906} C_DIS
LIN {X 0.050,Y -420.856,Z 1572.472,A 0.000,B 0.000,C 90.000,E1 85.008} C_DIS
LIN {X -0.173,Y -401.639,Z 1572.457,A 0.000,B 0.000,C 90.000,E1 82.299} C_DIS
LIN {X -0.087,Y -387.158,Z 1572.445,A 0.000,B 0.000,C 90.000,E1 80.038} C_DIS
LIN {X -0.196,Y -368.483,Z 1572.427,A 0.000,B 0.000,C 90.000,E1 76.881} C_DIS
LIN {X 0.114,Y -355.468,Z 1572.414,A 0.000,B 0.000,C 90.000,E1 74.464} C_DIS
LIN {X 0.040,Y -344.301,Z 1572.402,A 0.000,B 0.000,C 90.000,E1 72.362} C_DIS
LIN {X 0.103,Y -328.830,Z 1572.385,A 0.000,B 0.000,C 90.000,E1 69.263} C_DIS
LIN {X 0.059,Y -317.211,Z 1572.371,A 0.000,B 0.000,C 90.000,E1 66.741} C_DIS
LIN {X 0.063,Y -307.146,Z 1572.358,A 0.000,B 0.000,C 90.000,E1 64.485} C_DIS
LIN {X -0.139,Y -295.941,Z 1572.344,A 0.000,B 0.000,C 90.000,E1 61.897} C_DIS
LIN {X -0.044,Y -286.082,Z 1572.331,A 0.000,B 0.000,C 90.000,E1 59.537} C_DIS
LIN {X 0.061,Y -274.864,Z 1572.316,A 0.000,B 0.000,C 90.000,E1 56.786} C_DIS
LIN {X 0.033,Y -265.212,Z 1572.302,A 0.000,B 0.000,C 90.000,E1 54.356} C_DIS
LIN {X -0.025,Y -252.989,Z 1572.284,A 0.000,B 0.000,C 90.000,E1 51.170} C_DIS
LIN {X 0.054,Y -241.601,Z 1572.266,A 0.000,B 0.000,C 90.000,E1 47.877} C_DIS
LIN {X 0.111,Y -231.192,Z 1572.247,A 0.000,B 0.000,C 90.000,E1 44.514} C_DIS
LIN {X -0.017,Y -222.743,Z 1572.231,A 0.000,B 0.000,C 90.000,E1 41.515} C_DIS
LIN {X -0.131,Y -215.060,Z 1572.214,A 0.000,B 0.000,C 90.000,E1 38.463} C_DIS
LIN {X -0.055,Y -208.146,Z 1572.196,A 0.000,B 0.000,C 90.000,E1 35.311} C_DIS
LIN {X -0.054,Y -201.996,Z 1572.178,A 0.000,B 0.000,C 90.000,E1 32.133} C_DIS
LIN {X -0.006,Y -196.653,Z 1572.161,A 0.000,B 0.000,C 90.000,E1 28.899} C_DIS
LIN {X -0.015,Y -192.050,Z 1572.142,A 0.000,B 0.000,C 90.000,E1 25.643} C_DIS
LIN {X -0.050,Y -187.203,Z 1572.120,A 0.000,B 0.000,C 90.000,E1 21.535} C_DIS
LIN {X 0.032,Y -183.157,Z 1572.096,A 0.000,B 0.000,C 90.000,E1 17.347} C_DIS
LIN {X 0.047,Y -179.379,Z 1572.068,A 0.000,B 0.000,C 90.000,E1 12.299} C_DIS
LIN {X 0.023,Y -176.226,Z 1572.035,A 0.000,B 0.000,C 90.000,E1 6.372} C_DIS
LIN {X -0.022,Y -174.195,Z 1571.993,A 0.000,B 0.000,C 90.000,E1 358.682} C_DIS
LIN {X -0.038,Y -175.673,Z 1571.940,A 0.000,B 0.000,C 90.000,E1 349.275} C_DIS
LIN {X -0.021,Y -178.326,Z 1571.912,A 0.000,B 0.000,C 90.000,E1 344.157} C_DIS
LIN {X -0.056,Y -181.665,Z 1571.888,A 0.000,B 0.000,C 90.000,E1 339.934} C_DIS
LIN {X -0.078,Y -186.050,Z 1571.865,A 0.000,B 0.000,C 90.000,E1 335.741} C_DIS
LIN {X -0.008,Y -191.457,Z 1571.842,A 0.000,B 0.000,C 90.000,E1 331.563} C_DIS
LIN {X -0.021,Y -196.537,Z 1571.824,A 0.000,B 0.000,C 90.000,E1 328.280} C_DIS
LIN {X 0.007,Y -202.384,Z 1571.806,A 0.000,B 0.000,C 90.000,E1 325.022} C_DIS
LIN {X -0.025,Y -209.069,Z 1571.788,A 0.000,B 0.000,C 90.000,E1 321.823} C_DIS
LIN {X 0.035,Y -216.628,Z 1571.770,A 0.000,B 0.000,C 90.000,E1 318.647} C_DIS
LIN {X 0.025,Y -225.999,Z 1571.751,A 0.000,B 0.000,C 90.000,E1 315.162} C_DIS
LIN {X 0.018,Y -235.301,Z 1571.734,A 0.000,B 0.000,C 90.000,E1 312.123} C_DIS
LIN {X 0.015,Y -241.675,Z 1571.724,A 0.000,B 0.000,C 90.000,E1 310.253} C_DIS
LIN {X 0.123,Y -247.389,Z 1571.715,A 0.000,B 0.000,C 90.000,E1 308.749} C_DIS
LIN {X -0.007,Y -253.901,Z 1571.707,A 0.000,B 0.000,C 90.000,E1 307.317} C_DIS
LIN {X 0.028,Y -265.093,Z 1571.695,A 0.000,B 0.000,C 90.000,E1 305.152} C_DIS
LIN {X 0.116,Y -275.479,Z 1571.686,A 0.000,B 0.000,C 90.000,E1 303.372} C_DIS
LIN {X -0.078,Y -291.753,Z 1571.672,A 0.000,B 0.000,C 90.000,E1 301.003} C_DIS
LIN {X -0.067,Y -309.037,Z 1571.659,A 0.000,B 0.000,C 90.000,E1 298.665} C_DIS
LIN {X 0.153,Y -321.595,Z 1571.650,A 0.000,B 0.000,C 90.000,E1 297.001} C_DIS
LIN {X -0.176,Y -336.671,Z 1571.640,A 0.000,B 0.000,C 90.000,E1 295.155} C_DIS
LIN {X 0.179,Y -354.049,Z 1571.628,A 0.000,B 0.000,C 90.000,E1 292.950} C_DIS
LIN {X -0.206,Y -369.519,Z 1571.618,A 0.000,B 0.000,C 90.000,E1 291.227} C_DIS
LIN {X -0.099,Y -382.190,Z 1571.610,A 0.000,B 0.000,C 90.000,E1 289.758} C_DIS
LIN {X -0.193,Y -389.393,Z 1571.605,A 0.000,B 0.000,C 90.000,E1 288.906} C_DIS
LIN {X 0.143,Y -396.044,Z 1571.600,A 0.000,B 0.000,C 90.000,E1 288.000} C_DIS
LIN {X 0.055,Y -401.989,Z 1571.595,A 0.000,B 0.000,C 90.000,E1 287.166} C_DIS
LIN {X 0.133,Y -407.237,Z 1571.591,A 0.000,B 0.000,C 90.000,E1 286.315} C_DIS
LIN {X 0.146,Y -411.563,Z 1571.586,A 0.000,B 0.000,C 90.000,E1 285.481} C_DIS
LIN {X 0.089,Y -415.052,Z 1571.582,A 0.000,B 0.000,C 90.000,E1 284.662} C_DIS
LIN {X 0.042,Y -416.944,Z 1571.578,A 0.000,B 0.000,C 90.000,E1 284.120} C_DIS
LIN {X -0.103,Y -418.402,Z 1571.575,A 0.000,B 0.000,C 90.000,E1 283.592} C_DIS
LIN {X 0.173,Y -419.497,Z 1571.572,A 0.000,B 0.000,C 90.000,E1 283.008} C_DIS
LIN {X 0.050,Y -420.110,Z 1571.569,A 0.000,B 0.000,C 90.000,E1 282.479} C_DIS
LIN {X -0.067,Y -420.274,Z 1571.566,A 0.000,B 0.000,C 90.000,E1 281.951} C_DIS
LIN {X -0.181,Y -419.902,Z 1571.563,A 0.000,B 0.000,C 90.000,E1 281.422} C_DIS
LIN {X 0.118,Y -419.021,Z 1571.560,A 0.000,B 0.000,C 90.000,E1 280.838} C_DIS
LIN {X 0.000,Y -417.557,Z 1571.557,A 0.000,B 0.000,C 90.000,E1 280.310} C_DIS
LIN {X -0.124,Y -415.452,Z 1571.554,A 0.000,B 0.000,C 90.000,E1 279.782} C_DIS
LIN {X 0.082,Y -412.682,Z 1571.551,A 0.000,B 0.000,C 90.000,E1 279.208} C_DIS
LIN {X -0.072,Y -409.190,Z 1571.548,A 0.000,B 0.000,C 90.000,E1 278.681} C_DIS
LIN {X 0.097,Y -404.916,Z 1571.545,A 0.000,B 0.000,C 90.000,E1 278.106} C_DIS
LIN {X -0.154,Y -399.860,Z 1571.542,A 0.000,B 0.000,C 90.000,E1 277.587} C_DIS
LIN {X 0.112,Y -394.038,Z 1571.539,A 0.000,B 0.000,C 90.000,E1 277.004} C_DIS
LIN {X -0.081,Y -388.118,Z 1571.536,A 0.000,B 0.000,C 90.000,E1 276.543} C_DIS
LIN {X -0.033,Y -381.964,Z 1571.534,A 0.000,B 0.000,C 90.000,E1 276.087} C_DIS
LIN {X -0.142,Y -372.680,Z 1571.531,A 0.000,B 0.000,C 90.000,E1 275.511} C_DIS
LIN {X -0.183,Y -362.951,Z 1571.528,A 0.000,B 0.000,C 90.000,E1 274.992} C_DIS
LIN {X 0.173,Y -353.372,Z 1571.525,A 0.000,B 0.000,C 90.000,E1 274.473} C_DIS
LIN {X -0.073,Y -340.528,Z 1571.522,A 0.000,B 0.000,C 90.000,E1 273.955} C_DIS
LIN {X -0.022,Y -327.630,Z 1571.519,A 0.000,B 0.000,C 90.000,E1 273.440} C_DIS
LIN {X -0.023,Y -317.455,Z 1571.517,A 0.000,B 0.000,C 90.000,E1 273.094} C_DIS
LIN {X -0.058,Y -307.361,Z 1571.516,A 0.000,B 0.000,C 90.000,E1 272.808} C_DIS
LIN {X 0.094,Y -296.399,Z 1571.514,A 0.000,B 0.000,C 90.000,E1 272.522} C_DIS
LIN {X -0.068,Y -284.237,Z 1571.513,A 0.000,B 0.000,C 90.000,E1 272.350} C_DIS
LIN {X 0.022,Y -266.498,Z 1571.512,A 0.000,B 0.000,C 90.000,E1 272.121} C_DIS
LIN {X 0.104,Y -254.412,Z 1571.511,A 0.000,B 0.000,C 90.000,E1 272.007} C_DIS
LIN {X 0.101,Y -239.333,Z 1571.511,A 0.000,B 0.000,C 90.000,E1 271.949} C_DIS
LIN {X 0.044,Y -181.267,Z 1571.511,A 0.000,B 0.000,C 90.000,E1 271.949} C_DIS
LIN {X -0.032,Y -181.580,Z 1571.501,A 0.000,B 0.000,C 90.000,E1 270.229} C_DIS
LIN {X -0.043,Y -180.892,Z 1571.473,A 0.000,B 0.000,C 90.000,E1 265.179} C_DIS
LIN {X -0.076,Y -179.243,Z 1571.450,A 0.000,B 0.000,C 90.000,E1 260.971} C_DIS
LIN {X -0.062,Y -178.645,Z 1571.440,A 0.000,B 0.000,C 90.000,E1 259.275} C_DIS
LIN {X 0.011,Y -175.696,Z 1571.412,A 0.000,B 0.000,C 90.000,E1 254.157} C_DIS
LIN {X 0.021,Y -172.412,Z 1571.388,A 0.000,B 0.000,C 90.000,E1 249.880} C_DIS
LIN {X 0.038,Y -171.228,Z 1571.379,A 0.000,B 0.000,C 90.000,E1 248.156} C_DIS
LIN {X 0.014,Y -167.508,Z 1571.355,A 0.000,B 0.000,C 90.000,E1 243.845} C_DIS
LIN {X -0.053,Y -166.904,Z 1571.350,A 0.000,B 0.000,C 90.000,E1 242.999} C_DIS
LIN {X -0.001,Y -162.212,Z 1571.321,A 0.000,B 0.000,C 90.000,E1 237.740} C_DIS
LIN {X -0.081,Y -160.790,Z 1571.311,A 0.000,B 0.000,C 90.000,E1 236.008} C_DIS
LIN {X 0.023,Y -157.580,Z 1571.291,A 0.000,B 0.000,C 90.000,E1 232.431} C_DIS
LIN {X 0.057,Y -155.612,Z 1571.276,A 0.000,B 0.000,C 90.000,E1 229.747} C_DIS
LIN {X 0.000,Y -151.891,Z 1571.252,A 0.000,B 0.000,C 90.000,E1 225.283} C_DIS
LIN {X -0.091,Y -150.119,Z 1571.237,A 0.000,B 0.000,C 90.000,E1 222.609} C_DIS
LIN {X 0.037,Y -146.911,Z 1571.211,A 0.000,B 0.000,C 90.000,E1 218.016} C_DIS
LIN {X -0.062,Y -145.498,Z 1571.196,A 0.000,B 0.000,C 90.000,E1 215.311} C_DIS
LIN {X 0.056,Y -142.904,Z 1571.171,A 0.000,B 0.000,C 90.000,E1 210.669} C_DIS
LIN {X -0.013,Y -141.524,Z 1571.150,A 0.000,B 0.000,C 90.000,E1 207.001} C_DIS
LIN {X 0.030,Y -139.396,Z 1571.114,A 0.000,B 0.000,C 90.000,E1 200.482} C_DIS
LIN {X 0.081,Y -139.109,Z 1571.104,A 0.000,B 0.000,C 90.000,E1 198.598} C_DIS
LIN {X -0.064,Y -138.353,Z 1571.057,A 0.000,B 0.000,C 90.000,E1 190.254} C_DIS
LIN {X 0.066,Y -139.510,Z 1571.005,A 0.000,B 0.000,C 90.000,E1 180.859} C_DIS
LIN {X 0.006,Y -141.151,Z 1570.974,A 0.000,B 0.000,C 90.000,E1 175.298} C_DIS
LIN {X -0.023,Y -142.532,Z 1570.958,A 0.000,B 0.000,C 90.000,E1 172.527} C_DIS
LIN {X 0.046,Y -144.799,Z 1570.933,A 0.000,B 0.000,C 90.000,E1 167.881} C_DIS
LIN {X 0.033,Y -147.418,Z 1570.912,A 0.000,B 0.000,C 90.000,E1 164.212} C_DIS
LIN {X 0.062,Y -149.995,Z 1570.892,A 0.000,B 0.000,C 90.000,E1 160.550} C_DIS
LIN {X 0.071,Y -153.324,Z 1570.872,A 0.000,B 0.000,C 90.000,E1 156.922} C_DIS
LIN {X -0.018,Y -155.023,Z 1570.862,A 0.000,B 0.000,C 90.000,E1 155.153} C_DIS
LIN {X 0.004,Y -158.670,Z 1570.842,A 0.000,B 0.000,C 90.000,E1 151.563} C_DIS
LIN {X 0.087,Y -161.948,Z 1570.827,A 0.000,B 0.000,C 90.000,E1 148.869} C_DIS
LIN {X -0.029,Y -166.139,Z 1570.808,A 0.000,B 0.000,C 90.000,E1 145.388} C_DIS
LIN {X -0.033,Y -171.151,Z 1570.788,A 0.000,B 0.000,C 90.000,E1 141.904} C_DIS
LIN {X 0.003,Y -176.030,Z 1570.769,A 0.000,B 0.000,C 90.000,E1 138.447} C_DIS
LIN {X -0.002,Y -180.282,Z 1570.755,A 0.000,B 0.000,C 90.000,E1 135.891} C_DIS
LIN {X -0.030,Y -185.696,Z 1570.736,A 0.000,B 0.000,C 90.000,E1 132.528} C_DIS
LIN {X 0.022,Y -190.299,Z 1570.722,A 0.000,B 0.000,C 90.000,E1 130.011} C_DIS
LIN {X 0.070,Y -197.626,Z 1570.699,A 0.000,B 0.000,C 90.000,E1 125.884} C_DIS
LIN {X 0.000,Y -200.884,Z 1570.690,A 0.000,B 0.000,C 90.000,E1 124.278} C_DIS
LIN {X -0.045,Y -203.959,Z 1570.681,A 0.000,B 0.000,C 90.000,E1 122.546} C_DIS
LIN {X -0.105,Y -320.759,Z 1570.681,A 0.000,B 0.000,C 90.000,E1 122.546} C_DIS
LIN {X 0.071,Y -323.123,Z 1570.680,A 0.000,B 0.000,C 90.000,E1 122.467} C_DIS
LIN {X 0.036,Y -328.574,Z 1570.679,A 0.000,B 0.000,C 90.000,E1 122.163} C_DIS
LIN {X -0.103,Y -331.546,Z 1570.677,A 0.000,B 0.000,C 90.000,E1 121.878} C_DIS
LIN {X -0.106,Y -333.544,Z 1570.675,A 0.000,B 0.000,C 90.000,E1 121.592} C_DIS
LIN {X 0.175,Y -335.109,Z 1570.674,A 0.000,B 0.000,C 90.000,E1 121.258} C_DIS
LIN {X 0.087,Y -342.704,Z 1570.663,A 0.000,B 0.000,C 90.000,E1 119.411} C_DIS
LIN {X 0.054,Y -355.023,Z 1570.648,A 0.000,B 0.000,C 90.000,E1 116.668} C_DIS
LIN {X 0.212,Y -368.825,Z 1570.633,A 0.000,B 0.000,C 90.000,E1 113.951} C_DIS
LIN {X 0.000,Y -382.432,Z 1570.620,A 0.000,B 0.000,C 90.000,E1 111.642} C_DIS
LIN {X 0.196,Y -397.396,Z 1570.608,A 0.000,B 0.000,C 90.000,E1 109.322} C_DIS
LIN {X 0.137,Y -413.821,Z 1570.595,A 0.000,B 0.000,C 90.000,E1 107.094} C_DIS
LIN {X -0.163,Y -431.821,Z 1570.583,A 0.000,B 0.000,C 90.000,E1 104.954} C_DIS
LIN {X -0.011,Y -451.354,Z 1570.571,A 0.000,B 0.000,C 90.000,E1 102.827} C_DIS
LIN {X -0.126,Y -471.593,Z 1570.560,A 0.000,B 0.000,C 90.000,E1 100.894} C_DIS
LIN {X -0.053,Y -492.348,Z 1570.551,A 0.000,B 0.000,C 90.000,E1 99.095} C_DIS
LIN {X 0.144,Y -494.723,Z 1570.549,A 0.000,B 0.000,C 90.000,E1 98.859} C_DIS
LIN {X -0.149,Y -496.522,Z 1570.548,A 0.000,B 0.000,C 90.000,E1 98.681} C_DIS
LIN {X 0.185,Y -498.098,Z 1570.547,A 0.000,B 0.000,C 90.000,E1 98.398} C_DIS
LIN {X 0.101,Y -499.273,Z 1570.545,A 0.000,B 0.000,C 90.000,E1 98.163} C_DIS
LIN {X -0.123,Y -500.673,Z 1570.543,A 0.000,B 0.000,C 90.000,E1 97.701} C_DIS
LIN {X 0.158,Y -501.016,Z 1570.540,A 0.000,B 0.000,C 90.000,E1 97.182} C_DIS
LIN {X -0.050,Y -500.358,Z 1570.537,A 0.000,B 0.000,C 90.000,E1 96.720} C_DIS
LIN {X 0.240,Y -498.592,Z 1570.535,A 0.000,B 0.000,C 90.000,E1 96.201} C_DIS
LIN {X 0.162,Y -497.190,Z 1570.533,A 0.000,B 0.000,C 90.000,E1 95.967} C_DIS
LIN {X -0.215,Y -481.036,Z 1570.520,A 0.000,B 0.000,C 90.000,E1 93.555} C_DIS
LIN {X 0.191,Y -471.185,Z 1570.511,A 0.000,B 0.000,C 90.000,E1 92.007} C_DIS
LIN {X 0.161,Y -462.659,Z 1570.504,A 0.000,B 0.000,C 90.000,E1 90.745} C_DIS
LIN {X -0.003,Y -453.717,Z 1570.497,A 0.000,B 0.000,C 90.000,E1 89.484} C_DIS
LIN {X 0.173,Y -444.384,Z 1570.490,A 0.000,B 0.000,C 90.000,E1 88.165} C_DIS
LIN {X -0.063,Y -432.624,Z 1570.481,A 0.000,B 0.000,C 90.000,E1 86.617} C_DIS
LIN {X 0.206,Y -416.776,Z 1570.469,A 0.000,B 0.000,C 90.000,E1 84.432} C_DIS
LIN {X -0.063,Y -396.029,Z 1570.452,A 0.000,B 0.000,C 90.000,E1 81.432} C_DIS
LIN {X 0.054,Y -374.978,Z 1570.433,A 0.000,B 0.000,C 90.000,E1 77.993} C_DIS
LIN {X 0.086,Y -361.805,Z 1570.420,A 0.000,B 0.000,C 90.000,E1 75.644} C_DIS
LIN {X -0.023,Y -348.955,Z 1570.407,A 0.000,B 0.000,C 90.000,E1 73.268} C_DIS
LIN {X 0.196,Y -336.281,Z 1570.393,A 0.000,B 0.000,C 90.000,E1 70.786} C_DIS
LIN {X 0.081,Y -319.956,Z 1570.374,A 0.000,B 0.000,C 90.000,E1 67.358} C_DIS
LIN {X 0.148,Y -309.871,Z 1570.362,A 0.000,B 0.000,C 90.000,E1 65.101} C_DIS
LIN {X 0.159,Y -297.146,Z 1570.345,A 0.000,B 0.000,C 90.000,E1 62.153} C_DIS
LIN {X -0.110,Y -288.703,Z 1570.334,A 0.000,B 0.000,C 90.000,E1 60.205} C_DIS
LIN {X 0.063,Y -277.441,Z 1570.319,A 0.000,B 0.000,C 90.000,E1 57.454} C_DIS
LIN {X -0.056,Y -267.810,Z 1570.306,A 0.000,B 0.000,C 90.000,E1 55.055} C_DIS
LIN {X 0.080,Y -258.239,Z 1570.292,A 0.000,B 0.000,C 90.000,E1 52.557} C_DIS
LIN {X -0.017,Y -246.486,Z 1570.274,A 0.000,B 0.000,C 90.000,E1 49.337} C_DIS
LIN {X -0.152,Y -235.711,Z 1570.256,A 0.000,B 0.000,C 90.000,E1 46.053} C_DIS
LIN {X -0.015,Y -226.888,Z 1570.239,A 0.000,B 0.000,C 90.000,E1 43.014} C_DIS
LIN {X 0.091,Y -218.852,Z 1570.222,A 0.000,B 0.000,C 90.000,E1 39.930} C_DIS
LIN {X -0.085,Y -211.552,Z 1570.205,A 0.000,B 0.000,C 90.000,E1 36.870} C_DIS
LIN {X -0.052,Y -205.089,Z 1570.187,A 0.000,B 0.000,C 90.000,E1 33.706} C_DIS
LIN {X 0.102,Y -199.328,Z 1570.169,A 0.000,B 0.000,C 90.000,E1 30.463} C_DIS
LIN {X -0.014,Y -194.407,Z 1570.151,A 0.000,B 0.000,C 90.000,E1 27.257} C_DIS
LIN {X 0.005,Y -189.189,Z 1570.129,A 0.000,B 0.000,C 90.000,E1 23.153} C_DIS
LIN {X -0.073,Y -184.880,Z 1570.106,A 0.000,B 0.000,C 90.000,E1 19.033} C_DIS
LIN {X -0.004,Y -181.341,Z 1570.082,A 0.000,B 0.000,C 90.000,E1 14.828} C_DIS
LIN {X -0.057,Y -178.085,Z 1570.054,A 0.000,B 0.000,C 90.000,E1 9.782} C_DIS
LIN {X 0.065,Y -175.735,Z 1570.026,A 0.000,B 0.000,C 90.000,E1 4.645} C_DIS
LIN {X 0.069,Y -174.590,Z 1569.969,A 0.000,B 0.000,C 90.000,E1 354.375} C_DIS
LIN {X -0.083,Y -176.685,Z 1569.931,A 0.000,B 0.000,C 90.000,E1 347.589} C_DIS
LIN {X -0.081,Y -179.786,Z 1569.903,A 0.000,B 0.000,C 90.000,E1 342.489} C_DIS
LIN {X 0.045,Y -183.557,Z 1569.879,A 0.000,B 0.000,C 90.000,E1 338.230} C_DIS
LIN {X -0.039,Y -188.320,Z 1569.856,A 0.000,B 0.000,C 90.000,E1 334.076} C_DIS
LIN {X 0.032,Y -194.095,Z 1569.833,A 0.000,B 0.000,C 90.000,E1 329.921} C_DIS
LIN {X 0.121,Y -199.517,Z 1569.815,A 0.000,B 0.000,C 90.000,E1 326.628} C_DIS
LIN {X 0.064,Y -205.762,Z 1569.797,A 0.000,B 0.000,C 90.000,E1 323.417} C_DIS
LIN {X -0.090,Y -212.819,Z 1569.779,A 0.000,B 0.000,C 90.000,E1 320.275} C_DIS
LIN {X -0.117,Y -220.722,Z 1569.762,A 0.000,B 0.000,C 90.000,E1 317.148} C_DIS
LIN {X 0.060,Y -229.362,Z 1569.745,A 0.000,B 0.000,C 90.000,E1 314.028} C_DIS
LIN {X -0.004,Y -238.986,Z 1569.728,A 0.000,B 0.000,C 90.000,E1 311.024} C_DIS
LIN {X -0.126,Y -245.833,Z 1569.718,A 0.000,B 0.000,C 90.000,E1 309.197} C_DIS
LIN {X -0.127,Y -252.091,Z 1569.709,A 0.000,B 0.000,C 90.000,E1 307.729} C_DIS
LIN {X 0.037,Y -261.076,Z 1569.699,A 0.000,B 0.000,C 90.000,E1 305.884} C_DIS
LIN {X -0.010,Y -271.025,Z 1569.690,A 0.000,B 0.000,C 90.000,E1 304.119} C_DIS
LIN {X 0.172,Y -282.094,Z 1569.680,A 0.000,B 0.000,C 90.000,E1 302.339} C_DIS
LIN {X -0.020,Y -301.373,Z 1569.665,A 0.000,B 0.000,C 90.000,E1 299.667} C_DIS
LIN {X -0.079,Y -316.274,Z 1569.654,A 0.000,B 0.000,C 90.000,E1 297.719} C_DIS
LIN {X -0.070,Y -331.409,Z 1569.643,A 0.000,B 0.000,C 90.000,E1 295.796} C_DIS
LIN {X 0.093,Y -343.888,Z 1569.635,A 0.000,B 0.000,C 90.000,E1 294.207} C_DIS
LIN {X -0.045,Y -366.712,Z 1569.620,A 0.000,B 0.000,C 90.000,E1 291.535} C_DIS
LIN {X -0.041,Y -379.627,Z 1569.611,A 0.000,B 0.000,C 90.000,E1 290.066} C_DIS
LIN {X -0.155,Y -387.048,Z 1569.607,A 0.000,B 0.000,C 90.000,E1 289.214} C_DIS
LIN {X -0.206,Y -393.926,Z 1569.602,A 0.000,B 0.000,C 90.000,E1 288.362} C_DIS
LIN {X 0.176,Y -400.143,Z 1569.597,A 0.000,B 0.000,C 90.000,E1 287.457} C_DIS
LIN {X 0.127,Y -405.716,Z 1569.592,A 0.000,B 0.000,C 90.000,E1 286.622} C_DIS
LIN {X 0.124,Y -410.380,Z 1569.588,A 0.000,B 0.000,C 90.000,E1 285.788} C_DIS
LIN {X 0.168,Y -414.191,Z 1569.583,A 0.000,B 0.000,C 90.000,E1 284.954} C_DIS
LIN {X -0.162,Y -417.192,Z 1569.579,A 0.000,B 0.000,C 90.000,E1 284.175} C_DIS
LIN {X 0.100,Y -418.726,Z 1569.576,A 0.000,B 0.000,C 90.000,E1 283.592} C_DIS
LIN {X -0.032,Y -419.854,Z 1569.573,A 0.000,B 0.000,C 90.000,E1 283.063} C_DIS
LIN {X -0.155,Y -420.542,Z 1569.570,A 0.000,B 0.000,C 90.000,E1 282.535} C_DIS
LIN {X 0.143,Y -420.731,Z 1569.567,A 0.000,B 0.000,C 90.000,E1 281.951} C_DIS
LIN {X 0.031,Y -420.383,Z 1569.563,A 0.000,B 0.000,C 90.000,E1 281.422} C_DIS
LIN {X -0.080,Y -419.574,Z 1569.560,A 0.000,B 0.000,C 90.000,E1 280.894} C_DIS
LIN {X 0.216,Y -418.175,Z 1569.557,A 0.000,B 0.000,C 90.000,E1 280.310} C_DIS
LIN {X 0.023,Y -416.120,Z 1569.554,A 0.000,B 0.000,C 90.000,E1 279.792} C_DIS
LIN {X -0.105,Y -413.465,Z 1569.551,A 0.000,B 0.000,C 90.000,E1 279.265} C_DIS
LIN {X 0.089,Y -410.012,Z 1569.548,A 0.000,B 0.000,C 90.000,E1 278.690} C_DIS
LIN {X -0.079,Y -405.814,Z 1569.545,A 0.000,B 0.000,C 90.000,E1 278.163} C_DIS
LIN {X 0.073,Y -400.791,Z 1569.542,A 0.000,B 0.000,C 90.000,E1 277.587} C_DIS
LIN {X -0.109,Y -395.029,Z 1569.539,A 0.000,B 0.000,C 90.000,E1 277.068} C_DIS
LIN {X 0.071,Y -389.068,Z 1569.536,A 0.000,B 0.000,C 90.000,E1 276.549} C_DIS
LIN {X 0.161,Y -382.977,Z 1569.534,A 0.000,B 0.000,C 90.000,E1 276.087} C_DIS
LIN {X 0.052,Y -373.685,Z 1569.531,A 0.000,B 0.000,C 90.000,E1 275.511} C_DIS
LIN {X -0.018,Y -363.937,Z 1569.528,A 0.000,B 0.000,C 90.000,E1 274.992} C_DIS
LIN {X 0.150,Y -351.130,Z 1569.524,A 0.000,B 0.000,C 90.000,E1 274.359} C_DIS
LIN {X -0.032,Y -338.271,Z 1569.521,A 0.000,B 0.000,C 90.000,E1 273.841} C_DIS
LIN {X 0.067,Y -325.165,Z 1569.519,A 0.000,B 0.000,C 90.000,E1 273.326} C_DIS
LIN {X 0.156,Y -315.129,Z 1569.517,A 0.000,B 0.000,C 90.000,E1 272.980} C_DIS
LIN {X 0.148,Y -304.721,Z 1569.515,A 0.000,B 0.000,C 90.000,E1 272.694} C_DIS
LIN {X 0.101,Y -293.694,Z 1569.514,A 0.000,B 0.000,C 90.000,E1 272.465} C_DIS
LIN {X -0.022,Y -280.512,Z 1569.513,A 0.000,B 0.000,C 90.000,E1 272.293} C_DIS
LIN {X 0.045,Y -267.090,Z 1569.512,A 0.000,B 0.000,C 90.000,E1 272.121} C_DIS
LIN {X 0.114,Y -254.117,Z 1569.511,A 0.000,B 0.000,C 90.000,E1 272.007} C_DIS
LIN {X -0.091,Y -242.724,Z 1569.511,A 0.000,B 0.000,C 90.000,E1 272.007} C_DIS
LIN {X -0.090,Y -181.265,Z 1569.511,A 0.000,B 0.000,C 90.000,E1 272.007} C_DIS
LIN {X 0.049,Y -181.581,Z 1569.501,A 0.000,B 0.000,C 90.000,E1 270.229} C_DIS
LIN {X 0.038,Y -180.895,Z 1569.473,A 0.000,B 0.000,C 90.000,E1 265.179} C_DIS
LIN {X 0.045,Y -179.836,Z 1569.459,A 0.000,B 0.000,C 90.000,E1 262.648} C_DIS
LIN {X -0.076,Y -179.023,Z 1569.445,A 0.000,B 0.000,C 90.000,E1 260.151} C_DIS
LIN {X -0.015,Y -178.663,Z 1569.440,A 0.000,B 0.000,C 90.000,E1 259.285} C_DIS
LIN {X 0.092,Y -175.713,Z 1569.412,A 0.000,B 0.000,C 90.000,E1 254.157} C_DIS
LIN {X -0.061,Y -172.429,Z 1569.388,A 0.000,B 0.000,C 90.000,E1 249.934} C_DIS
LIN {X -0.042,Y -171.255,Z 1569.379,A 0.000,B 0.000,C 90.000,E1 248.209} C_DIS
LIN {X -0.059,Y -167.528,Z 1569.355,A 0.000,B 0.000,C 90.000,E1 243.896} C_DIS
LIN {X 0.024,Y -166.922,Z 1569.350,A 0.000,B 0.000,C 90.000,E1 242.999} C_DIS
LIN {X -0.053,Y -162.918,Z 1569.326,A 0.000,B 0.000,C 90.000,E1 238.663} C_DIS
LIN {X -0.076,Y -161.592,Z 1569.316,A 0.000,B 0.000,C 90.000,E1 236.914} C_DIS
LIN {X 0.050,Y -158.333,Z 1569.296,A 0.000,B 0.000,C 90.000,E1 233.336} C_DIS
LIN {X 0.031,Y -155.636,Z 1569.277,A 0.000,B 0.000,C 90.000,E1 229.784} C_DIS
LIN {X -0.034,Y -151.909,Z 1569.252,A 0.000,B 0.000,C 90.000,E1 225.324} C_DIS
LIN {X -0.019,Y -150.142,Z 1569.237,A 0.000,B 0.000,C 90.000,E1 222.609} C_DIS
LIN {X 0.018,Y -146.928,Z 1569.211,A 0.000,B 0.000,C 90.000,E1 218.051} C_DIS
LIN {X 0.009,Y -145.516,Z 1569.196,A 0.000,B 0.000,C 90.000,E1 215.311} C_DIS
LIN {X 0.004,Y -142.916,Z 1569.171,A 0.000,B 0.000,C 90.000,E1 210.718} C_DIS
LIN {X 0.057,Y -141.538,Z 1569.150,A 0.000,B 0.000,C 90.000,E1 207.001} C_DIS
LIN {X -0.031,Y -139.402,Z 1569.114,A 0.000,B 0.000,C 90.000,E1 200.536} C_DIS
LIN {X -0.026,Y -139.117,Z 1569.104,A 0.000,B 0.000,C 90.000,E1 198.671} C_DIS
LIN {X 0.006,Y -138.353,Z 1569.057,A 0.000,B 0.000,C 90.000,E1 190.254} C_DIS
LIN {X -0.005,Y -139.505,Z 1569.005,A 0.000,B 0.000,C 90.000,E1 180.917} C_DIS
LIN {X -0.064,Y -141.140,Z 1568.974,A 0.000,B 0.000,C 90.000,E1 175.355} C_DIS
LIN {X 0.030,Y -142.519,Z 1568.959,A 0.000,B 0.000,C 90.000,E1 172.534} C_DIS
LIN {X -0.025,Y -144.782,Z 1568.933,A 0.000,B 0.000,C 90.000,E1 167.937} C_DIS
LIN {X -0.036,Y -147.398,Z 1568.912,A 0.000,B 0.000,C 90.000,E1 164.267} C_DIS
LIN {X -0.006,Y -149.972,Z 1568.892,A 0.000,B 0.000,C 90.000,E1 160.604} C_DIS
LIN {X 0.004,Y -153.294,Z 1568.872,A 0.000,B 0.000,C 90.000,E1 156.975} C_DIS
LIN {X -0.009,Y -154.998,Z 1568.862,A 0.000,B 0.000,C 90.000,E1 155.177} C_DIS
LIN {X 0.004,Y -158.639,Z 1568.842,A 0.000,B 0.000,C 90.000,E1 151.591} C_DIS
LIN {X -0.059,Y -161.914,Z 1568.827,A 0.000,B 0.000,C 90.000,E1 148.948} C_DIS
LIN {X 0.049,Y -166.104,Z 1568.808,A 0.000,B 0.000,C 90.000,E1 145.388} C_DIS
LIN {X 0.047,Y -171.113,Z 1568.788,A 0.000,B 0.000,C 90.000,E1 141.904} C_DIS
LIN {X -0.034,Y -175.989,Z 1568.769,A 0.000,B 0.000,C 90.000,E1 138.485} C_DIS
LIN {X 0.080,Y -180.236,Z 1568.755,A 0.000,B 0.000,C 90.000,E1 135.891} C_DIS
LIN {X 0.053,Y -185.651,Z 1568.736,A 0.000,B 0.000,C 90.000,E1 132.528} C_DIS
LIN {X 0.107,Y -190.250,Z 1568.722,A 0.000,B 0.000,C 90.000,E1 130.011} C_DIS
LIN {X -0.003,Y -197.578,Z 1568.700,A 0.000,B 0.000,C 90.000,E1 125.931} C_DIS
LIN {X -0.078,Y -200.840,Z 1568.691,A 0.000,B 0.000,C 90.000,E1 124.326} C_DIS
LIN {X 0.098,Y -203.884,Z 1568.681,A 0.000,B 0.000,C 90.000,E1 122.546} C_DIS
LIN {X 0.103,Y -320.454,Z 1568.681,A 0.000,B 0.000,C 90.000,E1 122.546} C_DIS
LIN {X -0.137,Y -325.752,Z 1568.680,A 0.000,B 0.000,C 90.000,E1 122.418} C_DIS
LIN {X 0.072,Y -328.201,Z 1568.679,A 0.000,B 0.000,C 90.000,E1 122.212} C_DIS
LIN {X 0.039,Y -331.483,Z 1568.677,A 0.000,B 0.000,C 90.000,E1 121.878} C_DIS
LIN {X 0.045,Y -333.449,Z 1568.676,A 0.000,B 0.000,C 90.000,E1 121.592} C_DIS
LIN {X -0.126,Y -334.993,Z 1568.674,A 0.000,B 0.000,C 90.000,E1 121.337} C_DIS
LIN {X -0.046,Y -346.513,Z 1568.658,A 0.000,B 0.000,C 90.000,E1 118.537} C_DIS
LIN {X 0.013,Y -359.301,Z 1568.643,A 0.000,B 0.000,C 90.000,E1 115.796} C_DIS
LIN {X -0.036,Y -373.604,Z 1568.628,A 0.000,B 0.000,C 90.000,E1 113.131} C_DIS
LIN {X 0.074,Y -387.694,Z 1568.616,A 0.000,B 0.000,C 90.000,E1 110.791} C_DIS
LIN {X -0.098,Y -403.176,Z 1568.603,A 0.000,B 0.000,C 90.000,E1 108.544} C_DIS
LIN {X -0.021,Y -420.161,Z 1568.591,A 0.000,B 0.000,C 90.000,E1 106.315} C_DIS
LIN {X 0.246,Y -438.765,Z 1568.579,A 0.000,B 0.000,C 90.000,E1 104.120} C_DIS
LIN {X -0.162,Y -458.624,Z 1568.567,A 0.000,B 0.000,C 90.000,E1 102.119} C_DIS
LIN {X 0.109,Y -479.058,Z 1568.557,A 0.000,B 0.000,C 90.000,E1 100.197} C_DIS
LIN {X 0.101,Y -492.098,Z 1568.551,A 0.000,B 0.000,C 90.000,E1 99.095} C_DIS
LIN {X -0.190,Y -494.500,Z 1568.549,A 0.000,B 0.000,C 90.000,E1 98.916} C_DIS
LIN {X 0.004,Y -496.324,Z 1568.548,A 0.000,B 0.000,C 90.000,E1 98.681} C_DIS
LIN {X -0.155,Y -497.920,Z 1568.547,A 0.000,B 0.000,C 90.000,E1 98.454} C_DIS
LIN {X 0.253,Y -499.109,Z 1568.546,A 0.000,B 0.000,C 90.000,E1 98.163} C_DIS
LIN {X 0.029,Y -500.534,Z 1568.543,A 0.000,B 0.000,C 90.000,E1 97.701} C_DIS
LIN {X -0.188,Y -500.897,Z 1568.540,A 0.000,B 0.000,C 90.000,E1 97.239} C_DIS
LIN {X 0.101,Y -500.261,Z 1568.537,A 0.000,B 0.000,C 90.000,E1 96.720} C_DIS
LIN {X -0.106,Y -498.521,Z 1568.535,A 0.000,B 0.000,C 90.000,E1 96.258} C_DIS
LIN {X -0.185,Y -497.136,Z 1568.533,A 0.000,B 0.000,C 90.000,E1 96.024} C_DIS
LIN {X -0.073,Y -481.009,Z 1568.520,A 0.000,B 0.000,C 90.000,E1 93.555} C_DIS
LIN {X -0.141,Y -471.176,Z 1568.511,A 0.000,B 0.000,C 90.000,E1 92.064} C_DIS
LIN {X -0.166,Y -462.657,Z 1568.504,A 0.000,B 0.000,C 90.000,E1 90.802} C_DIS
LIN {X 0.130,Y -453.732,Z 1568.497,A 0.000,B 0.000,C 90.000,E1 89.484} C_DIS
LIN {X -0.154,Y -444.400,Z 1568.490,A 0.000,B 0.000,C 90.000,E1 88.224} C_DIS
LIN {X 0.065,Y -432.669,Z 1568.481,A 0.000,B 0.000,C 90.000,E1 86.617} C_DIS
LIN {X -0.085,Y -416.845,Z 1568.469,A 0.000,B 0.000,C 90.000,E1 84.489} C_DIS
LIN {X -0.021,Y -397.933,Z 1568.454,A 0.000,B 0.000,C 90.000,E1 81.724} C_DIS
LIN {X 0.131,Y -378.434,Z 1568.437,A 0.000,B 0.000,C 90.000,E1 78.578} C_DIS
LIN {X -0.123,Y -363.498,Z 1568.422,A 0.000,B 0.000,C 90.000,E1 75.992} C_DIS
LIN {X 0.160,Y -350.628,Z 1568.409,A 0.000,B 0.000,C 90.000,E1 73.559} C_DIS
LIN {X -0.016,Y -339.443,Z 1568.397,A 0.000,B 0.000,C 90.000,E1 71.456} C_DIS
LIN {X -0.018,Y -322.823,Z 1568.378,A 0.000,B 0.000,C 90.000,E1 68.028} C_DIS
LIN {X -0.007,Y -312.748,Z 1568.365,A 0.000,B 0.000,C 90.000,E1 65.793} C_DIS
LIN {X -0.069,Y -301.299,Z 1568.351,A 0.000,B 0.000,C 90.000,E1 63.204} C_DIS
LIN {X -0.004,Y -291.494,Z 1568.338,A 0.000,B 0.000,C 90.000,E1 60.873} C_DIS
LIN {X -0.152,Y -280.201,Z 1568.323,A 0.000,B 0.000,C 90.000,E1 58.201} C_DIS
LIN {X 0.106,Y -269.200,Z 1568.308,A 0.000,B 0.000,C 90.000,E1 55.388} C_DIS
LIN {X 0.110,Y -259.662,Z 1568.294,A 0.000,B 0.000,C 90.000,E1 52.924} C_DIS
LIN {X 0.038,Y -249.124,Z 1568.278,A 0.000,B 0.000,C 90.000,E1 50.070} C_DIS
LIN {X -0.011,Y -238.152,Z 1568.260,A 0.000,B 0.000,C 90.000,E1 46.782} C_DIS
LIN {X 0.006,Y -229.158,Z 1568.243,A 0.000,B 0.000,C 90.000,E1 43.785} C_DIS
LIN {X 0.002,Y -220.929,Z 1568.226,A 0.000,B 0.000,C 90.000,E1 40.744} C_DIS
LIN {X 0.006,Y -213.464,Z 1568.209,A 0.000,B 0.000,C 90.000,E1 37.649} C_DIS
LIN {X -0.087,Y -206.818,Z 1568.192,A 0.000,B 0.000,C 90.000,E1 34.532} C_DIS
LIN {X -0.058,Y -200.888,Z 1568.174,A 0.000,B 0.000,C 90.000,E1 31.337} C_DIS
LIN {X -0.037,Y -195.778,Z 1568.156,A 0.000,B 0.000,C 90.000,E1 28.103} C_DIS
LIN {X -0.066,Y -190.369,Z 1568.133,A 0.000,B 0.000,C 90.000,E1 24.027} C_DIS
LIN {X -0.040,Y -185.919,Z 1568.110,A 0.000,B 0.000,C 90.000,E1 19.885} C_DIS
LIN {X -0.059,Y -182.231,Z 1568.087,A 0.000,B 0.000,C 90.000,E1 15.717} C_DIS
LIN {X -0.039,Y -178.819,Z 1568.059,A 0.000,B 0.000,C 90.000,E1 10.658} C_DIS
LIN {X 0.009,Y -175.982,Z 1568.026,A 0.000,B 0.000,C 90.000,E1 4.702} C_DIS
LIN {X 0.045,Y -174.751,Z 1567.974,A 0.000,B 0.000,C 90.000,E1 355.241} C_DIS
LIN {X -0.061,Y -176.945,Z 1567.931,A 0.000,B 0.000,C 90.000,E1 347.589} C_DIS
LIN {X -0.048,Y -180.051,Z 1567.903,A 0.000,B 0.000,C 90.000,E1 342.489} C_DIS
LIN {X -0.084,Y -183.820,Z 1567.879,A 0.000,B 0.000,C 90.000,E1 338.284} C_DIS
LIN {X 0.010,Y -188.550,Z 1567.856,A 0.000,B 0.000,C 90.000,E1 334.076} C_DIS
LIN {X -0.085,Y -193.068,Z 1567.838,A 0.000,B 0.000,C 90.000,E1 330.795} C_DIS
LIN {X -0.028,Y -198.253,Z 1567.819,A 0.000,B 0.000,C 90.000,E1 327.502} C_DIS
LIN {X -0.067,Y -204.265,Z 1567.801,A 0.000,B 0.000,C 90.000,E1 324.276} C_DIS
LIN {X -0.099,Y -211.051,Z 1567.784,A 0.000,B 0.000,C 90.000,E1 321.090} C_DIS
LIN {X -0.012,Y -218.712,Z 1567.766,A 0.000,B 0.000,C 90.000,E1 317.919} C_DIS
LIN {X 0.051,Y -228.239,Z 1567.747,A 0.000,B 0.000,C 90.000,E1 314.433} C_DIS
LIN {X -0.060,Y -237.690,Z 1567.730,A 0.000,B 0.000,C 90.000,E1 311.434} C_DIS
LIN {X -0.026,Y -244.327,Z 1567.720,A 0.000,B 0.000,C 90.000,E1 309.564} C_DIS
LIN {X -0.044,Y -250.379,Z 1567.712,A 0.000,B 0.000,C 90.000,E1 308.096} C_DIS
LIN {X -0.110,Y -259.063,Z 1567.702,A 0.000,B 0.000,C 90.000,E1 306.297} C_DIS
LIN {X 0.020,Y -268.791,Z 1567.692,A 0.000,B 0.000,C 90.000,E1 304.485} C_DIS
LIN {X -0.059,Y -279.630,Z 1567.682,A 0.000,B 0.000,C 90.000,E1 302.752} C_DIS
LIN {X 0.081,Y -298.724,Z 1567.667,A 0.000,B 0.000,C 90.000,E1 300.001} C_DIS
LIN {X -0.051,Y -316.186,Z 1567.654,A 0.000,B 0.000,C 90.000,E1 297.719} C_DIS
LIN {X -0.041,Y -331.349,Z 1567.643,A 0.000,B 0.000,C 90.000,E1 295.796} C_DIS
LIN {X 0.122,Y -343.870,Z 1567.635,A 0.000,B 0.000,C 90.000,E1 294.207} C_DIS
LIN {X 0.069,Y -364.416,Z 1567.621,A 0.000,B 0.000,C 90.000,E1 291.791} C_DIS
LIN {X -0.039,Y -377.273,Z 1567.613,A 0.000,B 0.000,C 90.000,E1 290.355} C_DIS
LIN {X 0.196,Y -384.838,Z 1567.608,A 0.000,B 0.000,C 90.000,E1 289.450} C_DIS
LIN {X 0.121,Y -391.941,Z 1567.603,A 0.000,B 0.000,C 90.000,E1 288.598} C_DIS
LIN {X -0.006,Y -398.427,Z 1567.599,A 0.000,B 0.000,C 90.000,E1 287.764} C_DIS
LIN {X 0.039,Y -404.219,Z 1567.594,A 0.000,B 0.000,C 90.000,E1 286.913} C_DIS
LIN {X -0.070,Y -407.638,Z 1567.591,A 0.000,B 0.000,C 90.000,E1 286.370} C_DIS
LIN {X -0.167,Y -412.062,Z 1567.586,A 0.000,B 0.000,C 90.000,E1 285.552} C_DIS
LIN {X -0.114,Y -415.609,Z 1567.582,A 0.000,B 0.000,C 90.000,E1 284.717} C_DIS
LIN {X -0.160,Y -417.540,Z 1567.579,A 0.000,B 0.000,C 90.000,E1 284.175} C_DIS
LIN {X 0.103,Y -419.114,Z 1567.576,A 0.000,B 0.000,C 90.000,E1 283.592} C_DIS
LIN {X -0.025,Y -420.265,Z 1567.573,A 0.000,B 0.000,C 90.000,E1 283.063} C_DIS
LIN {X -0.145,Y -420.969,Z 1567.570,A 0.000,B 0.000,C 90.000,E1 282.535} C_DIS
LIN {X 0.153,Y -421.173,Z 1567.567,A 0.000,B 0.000,C 90.000,E1 281.951} C_DIS
LIN {X 0.044,Y -420.959,Z 1567.563,A 0.000,B 0.000,C 90.000,E1 281.422} C_DIS
LIN {X -0.064,Y -420.080,Z 1567.560,A 0.000,B 0.000,C 90.000,E1 280.894} C_DIS
LIN {X -0.176,Y -418.725,Z 1567.557,A 0.000,B 0.000,C 90.000,E1 280.366} C_DIS
LIN {X 0.046,Y -416.698,Z 1567.554,A 0.000,B 0.000,C 90.000,E1 279.792} C_DIS
LIN {X -0.080,Y -414.044,Z 1567.551,A 0.000,B 0.000,C 90.000,E1 279.265} C_DIS
LIN {X 0.117,Y -410.631,Z 1567.548,A 0.000,B 0.000,C 90.000,E1 278.690} C_DIS
LIN {X -0.047,Y -406.479,Z 1567.545,A 0.000,B 0.000,C 90.000,E1 278.163} C_DIS
LIN {X 0.109,Y -401.454,Z 1567.542,A 0.000,B 0.000,C 90.000,E1 277.587} C_DIS
LIN {X -0.054,Y -395.728,Z 1567.539,A 0.000,B 0.000,C 90.000,E1 277.068} C_DIS
LIN {X 0.144,Y -389.804,Z 1567.536,A 0.000,B 0.000,C 90.000,E1 276.549} C_DIS
LIN {X -0.139,Y -383.743,Z 1567.534,A 0.000,B 0.000,C 90.000,E1 276.144} C_DIS
LIN {X -0.183,Y -377.452,Z 1567.532,A 0.000,B 0.000,C 90.000,E1 275.739} C_DIS
LIN {X 0.009,Y -371.031,Z 1567.530,A 0.000,B 0.000,C 90.000,E1 275.334} C_DIS
LIN {X 0.109,Y -361.351,Z 1567.527,A 0.000,B 0.000,C 90.000,E1 274.821} C_DIS
LIN {X 0.054,Y -348.565,Z 1567.524,A 0.000,B 0.000,C 90.000,E1 274.245} C_DIS
LIN {X -0.032,Y -335.728,Z 1567.521,A 0.000,B 0.000,C 90.000,E1 273.726} C_DIS
LIN {X 0.156,Y -325.863,Z 1567.519,A 0.000,B 0.000,C 90.000,E1 273.326} C_DIS
LIN {X -0.062,Y -315.996,Z 1567.517,A 0.000,B 0.000,C 90.000,E1 273.037} C_DIS
LIN {X -0.083,Y -305.487,Z 1567.515,A 0.000,B 0.000,C 90.000,E1 272.751} C_DIS
LIN {X 0.145,Y -294.354,Z 1567.514,A 0.000,B 0.000,C 90.000,E1 272.465} C_DIS
LIN {X 0.015,Y -281.301,Z 1567.513,A 0.000,B 0.000,C 90.000,E1 272.293} C_DIS
LIN {X 0.061,Y -267.640,Z 1567.512,A 0.000,B 0.000,C 90.000,E1 272.121} C_DIS
LIN {X -0.124,Y -254.424,Z 1567.511,A 0.000,B 0.000,C 90.000,E1 272.064} C_DIS
LIN {X -0.070,Y -242.098,Z 1567.511,A 0.000,B 0.000,C 90.000,E1 272.007} C_DIS
LIN {X -0.073,Y -181.265,Z 1567.511,A 0.000,B 0.000,C 90.000,E1 272.007} C_DIS
LIN {X 0.083,Y -181.581,Z 1567.501,A 0.000,B 0.000,C 90.000,E1 270.229} C_DIS
LIN {X 0.073,Y -180.896,Z 1567.473,A 0.000,B 0.000,C 90.000,E1 265.179} C_DIS
LIN {X 0.079,Y -179.841,Z 1567.459,A 0.000,B 0.000,C 90.000,E1 262.648} C_DIS
LIN {X -0.043,Y -179.026,Z 1567.445,A 0.000,B 0.000,C 90.000,E1 260.151} C_DIS
LIN {X 0.019,Y -178.669,Z 1567.441,A 0.000,B 0.000,C 90.000,E1 259.285} C_DIS
LIN {X -0.044,Y -175.720,Z 1567.412,A 0.000,B 0.000,C 90.000,E1 254.212} C_DIS
LIN {X -0.027,Y -172.436,Z 1567.388,A 0.000,B 0.000,C 90.000,E1 249.934} C_DIS
LIN {X -0.073,Y -171.265,Z 1567.379,A 0.000,B 0.000,C 90.000,E1 248.230} C_DIS
LIN {X -0.026,Y -167.535,Z 1567.355,A 0.000,B 0.000,C 90.000,E1 243.896} C_DIS
LIN {X -0.012,Y -166.151,Z 1567.345,A 0.000,B 0.000,C 90.000,E1 242.153} C_DIS
LIN {X -0.022,Y -162.928,Z 1567.326,A 0.000,B 0.000,C 90.000,E1 238.663} C_DIS
LIN {X -0.044,Y -161.599,Z 1567.316,A 0.000,B 0.000,C 90.000,E1 236.914} C_DIS
LIN {X 0.081,Y -158.343,Z 1567.297,A 0.000,B 0.000,C 90.000,E1 233.336} C_DIS
LIN {X -0.057,Y -155.646,Z 1567.277,A 0.000,B 0.000,C 90.000,E1 229.828} C_DIS
LIN {X -0.004,Y -151.917,Z 1567.252,A 0.000,B 0.000,C 90.000,E1 225.324} C_DIS
LIN {X 0.011,Y -150.152,Z 1567.237,A 0.000,B 0.000,C 90.000,E1 222.609} C_DIS
LIN {X -0.068,Y -146.934,Z 1567.212,A 0.000,B 0.000,C 90.000,E1 218.096} C_DIS
LIN {X 0.039,Y -145.522,Z 1567.196,A 0.000,B 0.000,C 90.000,E1 215.311} C_DIS
LIN {X 0.033,Y -142.921,Z 1567.171,A 0.000,B 0.000,C 90.000,E1 210.718} C_DIS
LIN {X -0.040,Y -141.544,Z 1567.150,A 0.000,B 0.000,C 90.000,E1 207.052} C_DIS
LIN {X -0.051,Y -139.403,Z 1567.114,A 0.000,B 0.000,C 90.000,E1 200.556} C_DIS
LIN {X 0.003,Y -139.120,Z 1567.104,A 0.000,B 0.000,C 90.000,E1 198.671} C_DIS
LIN {X 0.034,Y -138.352,Z 1567.057,A 0.000,B 0.000,C 90.000,E1 190.254} C_DIS
LIN {X 0.024,Y -139.503,Z 1567.005,A 0.000,B 0.000,C 90.000,E1 180.917} C_DIS
LIN {X -0.034,Y -141.134,Z 1566.974,A 0.000,B 0.000,C 90.000,E1 175.355} C_DIS
LIN {X 0.059,Y -142.514,Z 1566.959,A 0.000,B 0.000,C 90.000,E1 172.534} C_DIS
LIN {X 0.006,Y -144.775,Z 1566.933,A 0.000,B 0.000,C 90.000,E1 167.937} C_DIS
LIN {X -0.045,Y -147.389,Z 1566.913,A 0.000,B 0.000,C 90.000,E1 164.283} C_DIS
LIN {X 0.016,Y -150.720,Z 1566.887,A 0.000,B 0.000,C 90.000,E1 159.699} C_DIS
LIN {X -0.043,Y -154.201,Z 1566.867,A 0.000,B 0.000,C 90.000,E1 156.102} C_DIS
LIN {X 0.026,Y -157.640,Z 1566.847,A 0.000,B 0.000,C 90.000,E1 152.487} C_DIS
LIN {X -0.027,Y -161.900,Z 1566.827,A 0.000,B 0.000,C 90.000,E1 148.948} C_DIS
LIN {X 0.081,Y -166.089,Z 1566.808,A 0.000,B 0.000,C 90.000,E1 145.388} C_DIS
LIN {X 0.079,Y -171.098,Z 1566.788,A 0.000,B 0.000,C 90.000,E1 141.904} C_DIS
LIN {X 0.000,Y -175.972,Z 1566.769,A 0.000,B 0.000,C 90.000,E1 138.485} C_DIS
LIN {X 0.114,Y -180.217,Z 1566.755,A 0.000,B 0.000,C 90.000,E1 135.891} C_DIS
LIN {X 0.088,Y -185.632,Z 1566.736,A 0.000,B 0.000,C 90.000,E1 132.528} C_DIS
LIN {X -0.126,Y -190.229,Z 1566.723,A 0.000,B 0.000,C 90.000,E1 130.092} C_DIS
LIN {X 0.033,Y -197.557,Z 1566.700,A 0.000,B 0.000,C 90.000,E1 125.931} C_DIS
LIN {X -0.043,Y -200.822,Z 1566.691,A 0.000,B 0.000,C 90.000,E1 124.326} C_DIS
LIN {X -0.051,Y -203.816,Z 1566.681,A 0.000,B 0.000,C 90.000,E1 122.625} C_DIS
LIN {X -0.130,Y -319.826,Z 1566.681,A 0.000,B 0.000,C 90.000,E1 122.625} C_DIS
LIN {X 0.162,Y -321.880,Z 1566.681,A 0.000,B 0.000,C 90.000,E1 122.546} C_DIS
LIN {X -0.078,Y -326.009,Z 1566.680,A 0.000,B 0.000,C 90.000,E1 122.418} C_DIS
LIN {X 0.132,Y -328.333,Z 1566.679,A 0.000,B 0.000,C 90.000,E1 122.212} C_DIS
LIN {X 0.099,Y -331.518,Z 1566.677,A 0.000,B 0.000,C 90.000,E1 121.878} C_DIS
LIN {X 0.068,Y -333.480,Z 1566.676,A 0.000,B 0.000,C 90.000,E1 121.592} C_DIS
LIN {X -0.140,Y -335.015,Z 1566.674,A 0.000,B 0.000,C 90.000,E1 121.337} C_DIS
LIN {X 0.111,Y -349.218,Z 1566.655,A 0.000,B 0.000,C 90.000,E1 117.897} C_DIS
LIN {X -0.069,Y -362.336,Z 1566.640,A 0.000,B 0.000,C 90.000,E1 115.207} C_DIS
LIN {X 0.151,Y -376.992,Z 1566.625,A 0.000,B 0.000,C 90.000,E1 112.514} C_DIS
LIN {X -0.147,Y -391.422,Z 1566.612,A 0.000,B 0.000,C 90.000,E1 110.248} C_DIS
LIN {X 0.157,Y -407.271,Z 1566.600,A 0.000,B 0.000,C 90.000,E1 107.946} C_DIS
LIN {X -0.175,Y -424.650,Z 1566.588,A 0.000,B 0.000,C 90.000,E1 105.788} C_DIS
LIN {X 0.224,Y -443.659,Z 1566.576,A 0.000,B 0.000,C 90.000,E1 103.592} C_DIS
LIN {X 0.147,Y -463.680,Z 1566.564,A 0.000,B 0.000,C 90.000,E1 101.591} C_DIS
LIN {X -0.155,Y -486.863,Z 1566.553,A 0.000,B 0.000,C 90.000,E1 99.557} C_DIS
LIN {X 0.080,Y -492.095,Z 1566.551,A 0.000,B 0.000,C 90.000,E1 99.095} C_DIS
LIN {X -0.212,Y -494.475,Z 1566.549,A 0.000,B 0.000,C 90.000,E1 98.916} C_DIS
LIN {X -0.017,Y -496.279,Z 1566.548,A 0.000,B 0.000,C 90.000,E1 98.681} C_DIS
LIN {X -0.176,Y -497.856,Z 1566.547,A 0.000,B 0.000,C 90.000,E1 98.454} C_DIS
LIN {X 0.232,Y -499.032,Z 1566.546,A 0.000,B 0.000,C 90.000,E1 98.163} C_DIS
LIN {X 0.008,Y -500.434,Z 1566.543,A 0.000,B 0.000,C 90.000,E1 97.701} C_DIS
LIN {X -0.209,Y -500.777,Z 1566.540,A 0.000,B 0.000,C 90.000,E1 97.239} C_DIS
LIN {X 0.078,Y -500.121,Z 1566.537,A 0.000,B 0.000,C 90.000,E1 96.720} C_DIS
LIN {X -0.129,Y -498.359,Z 1566.535,A 0.000,B 0.000,C 90.000,E1 96.258} C_DIS
LIN {X -0.207,Y -496.958,Z 1566.533,A 0.000,B 0.000,C 90.000,E1 96.024} C_DIS
LIN {X -0.100,Y -480.849,Z 1566.520,A 0.000,B 0.000,C 90.000,E1 93.555} C_DIS
LIN {X -0.171,Y -471.032,Z 1566.511,A 0.000,B 0.000,C 90.000,E1 92.064} C_DIS
LIN {X -0.197,Y -462.510,Z 1566.504,A 0.000,B 0.000,C 90.000,E1 90.802} C_DIS
LIN {X 0.098,Y -453.574,Z 1566.497,A 0.000,B 0.000,C 90.000,E1 89.484} C_DIS
LIN {X -0.188,Y -444.259,Z 1566.490,A 0.000,B 0.000,C 90.000,E1 88.224} C_DIS
LIN {X 0.029,Y -432.539,Z 1566.481,A 0.000,B 0.000,C 90.000,E1 86.617} C_DIS
LIN {X -0.121,Y -416.770,Z 1566.469,A 0.000,B 0.000,C 90.000,E1 84.489} C_DIS
LIN {X -0.057,Y -397.869,Z 1566.454,A 0.000,B 0.000,C 90.000,E1 81.724} C_DIS
LIN {X 0.069,Y -380.083,Z 1566.438,A 0.000,B 0.000,C 90.000,E1 78.870} C_DIS
LIN {X 0.210,Y -365.043,Z 1566.424,A 0.000,B 0.000,C 90.000,E1 76.228} C_DIS
LIN {X 0.083,Y -352.137,Z 1566.410,A 0.000,B 0.000,C 90.000,E1 73.866} C_DIS
LIN {X -0.058,Y -340.948,Z 1566.399,A 0.000,B 0.000,C 90.000,E1 71.764} C_DIS
LIN {X 0.020,Y -325.636,Z 1566.381,A 0.000,B 0.000,C 90.000,E1 68.646} C_DIS
LIN {X 0.027,Y -314.068,Z 1566.367,A 0.000,B 0.000,C 90.000,E1 66.102} C_DIS
LIN {X 0.070,Y -305.437,Z 1566.356,A 0.000,B 0.000,C 90.000,E1 64.152} C_DIS
LIN {X 0.092,Y -294.181,Z 1566.342,A 0.000,B 0.000,C 90.000,E1 61.513} C_DIS
LIN {X -0.112,Y -284.267,Z 1566.329,A 0.000,B 0.000,C 90.000,E1 59.203} C_DIS
LIN {X 0.100,Y -273.191,Z 1566.314,A 0.000,B 0.000,C 90.000,E1 56.421} C_DIS
LIN {X 0.045,Y -263.684,Z 1566.300,A 0.000,B 0.000,C 90.000,E1 53.989} C_DIS
LIN {X -0.053,Y -251.719,Z 1566.282,A 0.000,B 0.000,C 90.000,E1 50.803} C_DIS
LIN {X -0.022,Y -240.545,Z 1566.264,A 0.000,B 0.000,C 90.000,E1 47.514} C_DIS
LIN {X 0.064,Y -231.404,Z 1566.247,A 0.000,B 0.000,C 90.000,E1 44.514} C_DIS
LIN {X -0.055,Y -222.980,Z 1566.231,A 0.000,B 0.000,C 90.000,E1 41.515} C_DIS
LIN {X 0.006,Y -215.356,Z 1566.214,A 0.000,B 0.000,C 90.000,E1 38.418} C_DIS
LIN {X -0.079,Y -208.510,Z 1566.196,A 0.000,B 0.000,C 90.000,E1 35.311} C_DIS
LIN {X -0.068,Y -202.449,Z 1566.178,A 0.000,B 0.000,C 90.000,E1 32.133} C_DIS
LIN {X -0.009,Y -197.151,Z 1566.161,A 0.000,B 0.000,C 90.000,E1 28.899} C_DIS
LIN {X -0.002,Y -191.543,Z 1566.138,A 0.000,B 0.000,C 90.000,E1 24.823} C_DIS
LIN {X 0.053,Y -186.973,Z 1566.115,A 0.000,B 0.000,C 90.000,E1 20.684} C_DIS
LIN {X -0.060,Y -182.472,Z 1566.087,A 0.000,B 0.000,C 90.000,E1 15.717} C_DIS
LIN {X -0.031,Y -179.050,Z 1566.059,A 0.000,B 0.000,C 90.000,E1 10.658} C_DIS
LIN {X 0.026,Y -176.215,Z 1566.026,A 0.000,B 0.000,C 90.000,E1 4.702} C_DIS
LIN {X 0.053,Y -175.013,Z 1565.974,A 0.000,B 0.000,C 90.000,E1 355.241} C_DIS
LIN {X -0.038,Y -177.199,Z 1565.931,A 0.000,B 0.000,C 90.000,E1 347.589} C_DIS
LIN {X -0.016,Y -180.311,Z 1565.903,A 0.000,B 0.000,C 90.000,E1 342.489} C_DIS
LIN {X -0.044,Y -184.084,Z 1565.879,A 0.000,B 0.000,C 90.000,E1 338.284} C_DIS
LIN {X -0.021,Y -188.787,Z 1565.856,A 0.000,B 0.000,C 90.000,E1 334.101} C_DIS
LIN {X -0.028,Y -193.277,Z 1565.838,A 0.000,B 0.000,C 90.000,E1 330.795} C_DIS
LIN {X -0.071,Y -198.439,Z 1565.819,A 0.000,B 0.000,C 90.000,E1 327.533} C_DIS
LIN {X 0.003,Y -204.390,Z 1565.802,A 0.000,B 0.000,C 90.000,E1 324.276} C_DIS
LIN {X -0.022,Y -211.135,Z 1565.784,A 0.000,B 0.000,C 90.000,E1 321.090} C_DIS
LIN {X 0.069,Y -218.756,Z 1565.766,A 0.000,B 0.000,C 90.000,E1 317.919} C_DIS
LIN {X 0.137,Y -228.238,Z 1565.747,A 0.000,B 0.000,C 90.000,E1 314.433} C_DIS
LIN {X 0.029,Y -237.655,Z 1565.730,A 0.000,B 0.000,C 90.000,E1 311.434} C_DIS
LIN {X 0.064,Y -244.276,Z 1565.720,A 0.000,B 0.000,C 90.000,E1 309.564} C_DIS
LIN {X 0.048,Y -250.313,Z 1565.712,A 0.000,B 0.000,C 90.000,E1 308.096} C_DIS
LIN {X -0.015,Y -258.952,Z 1565.702,A 0.000,B 0.000,C 90.000,E1 306.297} C_DIS
LIN {X -0.106,Y -268.650,Z 1565.692,A 0.000,B 0.000,C 90.000,E1 304.532} C_DIS
LIN {X 0.039,Y -279.465,Z 1565.682,A 0.000,B 0.000,C 90.000,E1 302.752} C_DIS
LIN {X -0.078,Y -298.539,Z 1565.667,A 0.000,B 0.000,C 90.000,E1 300.050} C_DIS
LIN {X 0.051,Y -316.018,Z 1565.654,A 0.000,B 0.000,C 90.000,E1 297.719} C_DIS
LIN {X 0.116,Y -328.659,Z 1565.645,A 0.000,B 0.000,C 90.000,E1 296.104} C_DIS
LIN {X -0.080,Y -341.287,Z 1565.636,A 0.000,B 0.000,C 90.000,E1 294.567} C_DIS
LIN {X -0.176,Y -364.415,Z 1565.621,A 0.000,B 0.000,C 90.000,E1 291.844} C_DIS
LIN {X -0.005,Y -377.401,Z 1565.613,A 0.000,B 0.000,C 90.000,E1 290.355} C_DIS
LIN {X -0.019,Y -387.298,Z 1565.607,A 0.000,B 0.000,C 90.000,E1 289.214} C_DIS
LIN {X -0.065,Y -394.230,Z 1565.602,A 0.000,B 0.000,C 90.000,E1 288.362} C_DIS
LIN {X -0.060,Y -400.528,Z 1565.597,A 0.000,B 0.000,C 90.000,E1 287.511} C_DIS
LIN {X -0.111,Y -406.128,Z 1565.593,A 0.000,B 0.000,C 90.000,E1 286.677} C_DIS
LIN {X 0.184,Y -409.396,Z 1565.589,A 0.000,B 0.000,C 90.000,E1 286.079} C_DIS
LIN {X 0.212,Y -413.538,Z 1565.585,A 0.000,B 0.000,C 90.000,E1 285.245} C_DIS
LIN {X 0.051,Y -415.857,Z 1565.582,A 0.000,B 0.000,C 90.000,E1 284.717} C_DIS
LIN {X 0.007,Y -417.846,Z 1565.579,A 0.000,B 0.000,C 90.000,E1 284.175} C_DIS
LIN {X -0.134,Y -419.446,Z 1565.576,A 0.000,B 0.000,C 90.000,E1 283.647} C_DIS
LIN {X 0.146,Y -420.633,Z 1565.573,A 0.000,B 0.000,C 90.000,E1 283.063} C_DIS
LIN {X 0.028,Y -421.392,Z 1565.570,A 0.000,B 0.000,C 90.000,E1 282.535} C_DIS
LIN {X -0.082,Y -421.637,Z 1565.567,A 0.000,B 0.000,C 90.000,E1 282.007} C_DIS
LIN {X -0.190,Y -421.432,Z 1565.564,A 0.000,B 0.000,C 90.000,E1 281.478} C_DIS
LIN {X 0.116,Y -420.665,Z 1565.561,A 0.000,B 0.000,C 90.000,E1 280.894} C_DIS
LIN {X 0.007,Y -419.334,Z 1565.558,A 0.000,B 0.000,C 90.000,E1 280.366} C_DIS
LIN {X -0.179,Y -417.367,Z 1565.555,A 0.000,B 0.000,C 90.000,E1 279.849} C_DIS
LIN {X 0.108,Y -414.754,Z 1565.552,A 0.000,B 0.000,C 90.000,E1 279.265} C_DIS
LIN {X -0.168,Y -413.218,Z 1565.550,A 0.000,B 0.000,C 90.000,E1 279.029} C_DIS
LIN {X 0.024,Y -409.481,Z 1565.547,A 0.000,B 0.000,C 90.000,E1 278.454} C_DIS
LIN {X -0.204,Y -404.943,Z 1565.544,A 0.000,B 0.000,C 90.000,E1 277.936} C_DIS
LIN {X 0.039,Y -399.641,Z 1565.541,A 0.000,B 0.000,C 90.000,E1 277.352} C_DIS
LIN {X 0.037,Y -393.767,Z 1565.538,A 0.000,B 0.000,C 90.000,E1 276.834} C_DIS
LIN {X -0.038,Y -387.722,Z 1565.535,A 0.000,B 0.000,C 90.000,E1 276.372} C_DIS
LIN {X 0.159,Y -381.540,Z 1565.533,A 0.000,B 0.000,C 90.000,E1 275.910} C_DIS
LIN {X -0.182,Y -375.191,Z 1565.531,A 0.000,B 0.000,C 90.000,E1 275.568} C_DIS
LIN {X 0.153,Y -365.481,Z 1565.528,A 0.000,B 0.000,C 90.000,E1 274.992} C_DIS
LIN {X -0.022,Y -352.616,Z 1565.525,A 0.000,B 0.000,C 90.000,E1 274.416} C_DIS
LIN {X 0.174,Y -339.872,Z 1565.521,A 0.000,B 0.000,C 90.000,E1 273.841} C_DIS
LIN {X -0.042,Y -326.757,Z 1565.519,A 0.000,B 0.000,C 90.000,E1 273.383} C_DIS
LIN {X 0.071,Y -317.054,Z 1565.517,A 0.000,B 0.000,C 90.000,E1 273.037} C_DIS
LIN {X 0.021,Y -306.470,Z 1565.515,A 0.000,B 0.000,C 90.000,E1 272.751} C_DIS
LIN {X -0.040,Y -295.760,Z 1565.514,A 0.000,B 0.000,C 90.000,E1 272.522} C_DIS
LIN {X 0.111,Y -282.982,Z 1565.513,A 0.000,B 0.000,C 90.000,E1 272.293} C_DIS
LIN {X -0.126,Y -269.479,Z 1565.512,A 0.000,B 0.000,C 90.000,E1 272.178} C_DIS
LIN {X -0.055,Y -257.061,Z 1565.511,A 0.000,B 0.000,C 90.000,E1 272.064} C_DIS
LIN {X -0.011,Y -246.014,Z 1565.511,A 0.000,B 0.000,C 90.000,E1 272.007} C_DIS
LIN {X -0.039,Y -181.263,Z 1565.511,A 0.000,B 0.000,C 90.000,E1 272.007} C_DIS
LIN {X 0.040,Y -181.581,Z 1565.501,A 0.000,B 0.000,C 90.000,E1 270.229} C_DIS
LIN {X 0.029,Y -180.894,Z 1565.473,A 0.000,B 0.000,C 90.000,E1 265.179} C_DIS
LIN {X 0.036,Y -179.835,Z 1565.459,A 0.000,B 0.000,C 90.000,E1 262.648} C_DIS
LIN {X 0.091,Y -179.023,Z 1565.445,A 0.000,B 0.000,C 90.000,E1 260.095} C_DIS
LIN {X -0.023,Y -178.660,Z 1565.440,A 0.000,B 0.000,C 90.000,E1 259.285} C_DIS
LIN {X 0.083,Y -175.711,Z 1565.412,A 0.000,B 0.000,C 90.000,E1 254.157} C_DIS
LIN {X -0.069,Y -172.427,Z 1565.388,A 0.000,B 0.000,C 90.000,E1 249.934} C_DIS
LIN {X -0.051,Y -171.252,Z 1565.379,A 0.000,B 0.000,C 90.000,E1 248.209} C_DIS
LIN {X -0.067,Y -167.525,Z 1565.355,A 0.000,B 0.000,C 90.000,E1 243.896} C_DIS
LIN {X 0.016,Y -166.921,Z 1565.350,A 0.000,B 0.000,C 90.000,E1 242.999} C_DIS
LIN {X -0.062,Y -162.916,Z 1565.326,A 0.000,B 0.000,C 90.000,E1 238.663} C_DIS
LIN {X -0.084,Y -161.589,Z 1565.316,A 0.000,B 0.000,C 90.000,E1 236.914} C_DIS
LIN {X 0.042,Y -158.331,Z 1565.296,A 0.000,B 0.000,C 90.000,E1 233.336} C_DIS
LIN {X 0.022,Y -155.633,Z 1565.277,A 0.000,B 0.000,C 90.000,E1 229.784} C_DIS
LIN {X -0.043,Y -151.908,Z 1565.252,A 0.000,B 0.000,C 90.000,E1 225.324} C_DIS
LIN {X -0.028,Y -150.140,Z 1565.237,A 0.000,B 0.000,C 90.000,E1 222.609} C_DIS
LIN {X 0.010,Y -146.925,Z 1565.211,A 0.000,B 0.000,C 90.000,E1 218.051} C_DIS
LIN {X 0.002,Y -145.514,Z 1565.196,A 0.000,B 0.000,C 90.000,E1 215.311} C_DIS
LIN {X -0.004,Y -142.915,Z 1565.171,A 0.000,B 0.000,C 90.000,E1 210.718} C_DIS
LIN {X 0.049,Y -141.536,Z 1565.150,A 0.000,B 0.000,C 90.000,E1 207.001} C_DIS
LIN {X -0.039,Y -139.401,Z 1565.114,A 0.000,B 0.000,C 90.000,E1 200.536} C_DIS
LIN {X -0.034,Y -139.116,Z 1565.104,A 0.000,B 0.000,C 90.000,E1 198.671} C_DIS
LIN {X -0.002,Y -138.352,Z 1565.057,A 0.000,B 0.000,C 90.000,E1 190.254} C_DIS
LIN {X -0.012,Y -139.506,Z 1565.005,A 0.000,B 0.000,C 90.000,E1 180.917} C_DIS
LIN {X -0.071,Y -141.140,Z 1564.974,A 0.000,B 0.000,C 90.000,E1 175.355} C_DIS
LIN {X 0.022,Y -142.521,Z 1564.959,A 0.000,B 0.000,C 90.000,E1 172.534} C_DIS
LIN {X -0.032,Y -144.784,Z 1564.933,A 0.000,B 0.000,C 90.000,E1 167.937} C_DIS
LIN {X -0.044,Y -147.400,Z 1564.912,A 0.000,B 0.000,C 90.000,E1 164.267} C_DIS
LIN {X -0.014,Y -149.975,Z 1564.892,A 0.000,B 0.000,C 90.000,E1 160.604} C_DIS
LIN {X -0.004,Y -153.298,Z 1564.872,A 0.000,B 0.000,C 90.000,E1 156.975} C_DIS
LIN {X -0.016,Y -155.001,Z 1564.862,A 0.000,B 0.000,C 90.000,E1 155.177} C_DIS
LIN {X -0.004,Y -158.642,Z 1564.842,A 0.000,B 0.000,C 90.000,E1 151.591} C_DIS
LIN {X 0.016,Y -161.918,Z 1564.827,A 0.000,B 0.000,C 90.000,E1 148.918} C_DIS
LIN {X 0.041,Y -166.108,Z 1564.808,A 0.000,B 0.000,C 90.000,E1 145.388} C_DIS
LIN {X 0.038,Y -171.118,Z 1564.788,A 0.000,B 0.000,C 90.000,E1 141.904} C_DIS
LIN {X -0.043,Y -175.993,Z 1564.769,A 0.000,B 0.000,C 90.000,E1 138.485} C_DIS
LIN {X 0.071,Y -180.242,Z 1564.755,A 0.000,B 0.000,C 90.000,E1 135.891} C_DIS
LIN {X 0.045,Y -185.656,Z 1564.736,A 0.000,B 0.000,C 90.000,E1 132.528} C_DIS
LIN {X 0.097,Y -190.255,Z 1564.722,A 0.000,B 0.000,C 90.000,E1 130.011} C_DIS
LIN {X -0.013,Y -197.583,Z 1564.700,A 0.000,B 0.000,C 90.000,E1 125.931} C_DIS
LIN {X -0.088,Y -200.845,Z 1564.691,A 0.000,B 0.000,C 90.000,E1 124.326} C_DIS
LIN {X 0.059,Y -203.759,Z 1564.681,A 0.000,B 0.000,C 90.000,E1 122.625} C_DIS
LIN {X 0.041,Y -320.235,Z 1564.681,A 0.000,B 0.000,C 90.000,E1 122.625} C_DIS
LIN {X 0.111,Y -325.878,Z 1564.680,A 0.000,B 0.000,C 90.000,E1 122.418} C_DIS
LIN {X -0.045,Y -328.371,Z 1564.679,A 0.000,B 0.000,C 90.000,E1 122.260} C_DIS
LIN {X 0.024,Y -331.720,Z 1564.677,A 0.000,B 0.000,C 90.000,E1 121.878} C_DIS
LIN {X -0.052,Y -333.644,Z 1564.675,A 0.000,B 0.000,C 90.000,E1 121.592} C_DIS
LIN {X 0.156,Y -335.147,Z 1564.674,A 0.000,B 0.000,C 90.000,E1 121.258} C_DIS
LIN {X 0.078,Y -347.953,Z 1564.657,A 0.000,B 0.000,C 90.000,E1 118.180} C_DIS
LIN {X 0.034,Y -360.917,Z 1564.641,A 0.000,B 0.000,C 90.000,E1 115.463} C_DIS
LIN {X -0.131,Y -375.416,Z 1564.627,A 0.000,B 0.000,C 90.000,E1 112.823} C_DIS
LIN {X 0.023,Y -389.691,Z 1564.614,A 0.000,B 0.000,C 90.000,E1 110.482} C_DIS
LIN {X -0.105,Y -405.374,Z 1564.601,A 0.000,B 0.000,C 90.000,E1 108.236} C_DIS
LIN {X -0.097,Y -422.573,Z 1564.589,A 0.000,B 0.000,C 90.000,E1 106.024} C_DIS
LIN {X -0.194,Y -441.411,Z 1564.577,A 0.000,B 0.000,C 90.000,E1 103.883} C_DIS
LIN {X 0.003,Y -461.366,Z 1564.566,A 0.000,B 0.000,C 90.000,E1 101.827} C_DIS
LIN {X 0.111,Y -484.457,Z 1564.554,A 0.000,B 0.000,C 90.000,E1 99.726} C_DIS
LIN {X -0.092,Y -492.311,Z 1564.550,A 0.000,B 0.000,C 90.000,E1 99.095} C_DIS
LIN {X 0.105,Y -494.615,Z 1564.549,A 0.000,B 0.000,C 90.000,E1 98.859} C_DIS
LIN {X -0.188,Y -496.359,Z 1564.548,A 0.000,B 0.000,C 90.000,E1 98.681} C_DIS
LIN {X 0.145,Y -497.889,Z 1564.547,A 0.000,B 0.000,C 90.000,E1 98.398} C_DIS
LIN {X 0.061,Y -499.026,Z 1564.545,A 0.000,B 0.000,C 90.000,E1 98.163} C_DIS
LIN {X -0.163,Y -500.368,Z 1564.543,A 0.000,B 0.000,C 90.000,E1 97.701} C_DIS
LIN {X 0.116,Y -500.659,Z 1564.540,A 0.000,B 0.000,C 90.000,E1 97.182} C_DIS
LIN {X -0.093,Y -499.949,Z 1564.537,A 0.000,B 0.000,C 90.000,E1 96.720} C_DIS
LIN {X 0.195,Y -498.121,Z 1564.535,A 0.000,B 0.000,C 90.000,E1 96.201} C_DIS
LIN {X 0.115,Y -496.678,Z 1564.533,A 0.000,B 0.000,C 90.000,E1 95.967} C_DIS
LIN {X 0.042,Y -478.983,Z 1564.518,A 0.000,B 0.000,C 90.000,E1 93.269} C_DIS
LIN {X -0.045,Y -469.099,Z 1564.510,A 0.000,B 0.000,C 90.000,E1 91.776} C_DIS
LIN {X 0.130,Y -458.730,Z 1564.501,A 0.000,B 0.000,C 90.000,E1 90.229} C_DIS
LIN {X -0.088,Y -449.613,Z 1564.494,A 0.000,B 0.000,C 90.000,E1 88.969} C_DIS
LIN {X 0.029,Y -440.127,Z 1564.487,A 0.000,B 0.000,C 90.000,E1 87.650} C_DIS
LIN {X 0.148,Y -428.327,Z 1564.478,A 0.000,B 0.000,C 90.000,E1 86.045} C_DIS
LIN {X -0.071,Y -412.645,Z 1564.466,A 0.000,B 0.000,C 90.000,E1 83.913} C_DIS
LIN {X -0.152,Y -395.845,Z 1564.452,A 0.000,B 0.000,C 90.000,E1 81.432} C_DIS
LIN {X -0.077,Y -378.198,Z 1564.437,A 0.000,B 0.000,C 90.000,E1 78.578} C_DIS
LIN {X 0.023,Y -363.234,Z 1564.422,A 0.000,B 0.000,C 90.000,E1 75.936} C_DIS
LIN {X -0.046,Y -350.373,Z 1564.409,A 0.000,B 0.000,C 90.000,E1 73.559} C_DIS
LIN {X 0.106,Y -337.626,Z 1564.395,A 0.000,B 0.000,C 90.000,E1 71.094} C_DIS
LIN {X 0.080,Y -322.500,Z 1564.378,A 0.000,B 0.000,C 90.000,E1 67.975} C_DIS
LIN {X 0.129,Y -311.008,Z 1564.364,A 0.000,B 0.000,C 90.000,E1 65.409} C_DIS
LIN {X 0.036,Y -298.156,Z 1564.347,A 0.000,B 0.000,C 90.000,E1 62.487} C_DIS
LIN {X -0.072,Y -289.724,Z 1564.336,A 0.000,B 0.000,C 90.000,E1 60.511} C_DIS
LIN {X -0.053,Y -277.092,Z 1564.319,A 0.000,B 0.000,C 90.000,E1 57.454} C_DIS
LIN {X -0.021,Y -267.576,Z 1564.306,A 0.000,B 0.000,C 90.000,E1 55.022} C_DIS
LIN {X -0.040,Y -258.172,Z 1564.292,A 0.000,B 0.000,C 90.000,E1 52.557} C_DIS
LIN {X 0.030,Y -246.557,Z 1564.274,A 0.000,B 0.000,C 90.000,E1 49.299} C_DIS
LIN {X 0.076,Y -235.857,Z 1564.255,A 0.000,B 0.000,C 90.000,E1 45.972} C_DIS
LIN {X 0.041,Y -227.091,Z 1564.239,A 0.000,B 0.000,C 90.000,E1 42.975} C_DIS
LIN {X 0.001,Y -219.111,Z 1564.222,A 0.000,B 0.000,C 90.000,E1 39.930} C_DIS
LIN {X 0.004,Y -211.879,Z 1564.205,A 0.000,B 0.000,C 90.000,E1 36.824} C_DIS
LIN {X 0.049,Y -205.490,Z 1564.187,A 0.000,B 0.000,C 90.000,E1 33.658} C_DIS
LIN {X 0.044,Y -199.812,Z 1564.169,A 0.000,B 0.000,C 90.000,E1 30.463} C_DIS
LIN {X -0.059,Y -194.949,Z 1564.151,A 0.000,B 0.000,C 90.000,E1 27.257} C_DIS
LIN {X 0.061,Y -190.724,Z 1564.133,A 0.000,B 0.000,C 90.000,E1 23.951} C_DIS
LIN {X 0.088,Y -186.350,Z 1564.110,A 0.000,B 0.000,C 90.000,E1 19.812} C_DIS
LIN {X 0.010,Y -182.055,Z 1564.082,A 0.000,B 0.000,C 90.000,E1 14.828} C_DIS
LIN {X -0.048,Y -178.795,Z 1564.054,A 0.000,B 0.000,C 90.000,E1 9.792} C_DIS
LIN {X 0.013,Y -175.901,Z 1564.017,A 0.000,B 0.000,C 90.000,E1 2.980} C_DIS
LIN {X 0.060,Y -175.274,Z 1563.974,A 0.000,B 0.000,C 90.000,E1 355.241} C_DIS
LIN {X -0.016,Y -177.454,Z 1563.931,A 0.000,B 0.000,C 90.000,E1 347.589} C_DIS
LIN {X 0.016,Y -180.566,Z 1563.903,A 0.000,B 0.000,C 90.000,E1 342.489} C_DIS
LIN {X -0.003,Y -184.341,Z 1563.879,A 0.000,B 0.000,C 90.000,E1 338.284} C_DIS
LIN {X 0.028,Y -189.012,Z 1563.856,A 0.000,B 0.000,C 90.000,E1 334.101} C_DIS
LIN {X 0.028,Y -193.491,Z 1563.838,A 0.000,B 0.000,C 90.000,E1 330.795} C_DIS
LIN {X -0.007,Y -198.615,Z 1563.820,A 0.000,B 0.000,C 90.000,E1 327.533} C_DIS
LIN {X 0.073,Y -204.540,Z 1563.802,A 0.000,B 0.000,C 90.000,E1 324.276} C_DIS
LIN {X 0.053,Y -211.224,Z 1563.784,A 0.000,B 0.000,C 90.000,E1 321.090} C_DIS
LIN {X 0.003,Y -218.801,Z 1563.766,A 0.000,B 0.000,C 90.000,E1 317.957} C_DIS
LIN {X -0.108,Y -228.245,Z 1563.747,A 0.000,B 0.000,C 90.000,E1 314.514} C_DIS
LIN {X -0.047,Y -237.636,Z 1563.730,A 0.000,B 0.000,C 90.000,E1 311.472} C_DIS
LIN {X 0.147,Y -244.223,Z 1563.720,A 0.000,B 0.000,C 90.000,E1 309.564} C_DIS
LIN {X 0.133,Y -250.262,Z 1563.712,A 0.000,B 0.000,C 90.000,E1 308.096} C_DIS
LIN {X 0.071,Y -258.858,Z 1563.702,A 0.000,B 0.000,C 90.000,E1 306.297} C_DIS
LIN {X -0.017,Y -268.536,Z 1563.692,A 0.000,B 0.000,C 90.000,E1 304.532} C_DIS
LIN {X 0.128,Y -279.321,Z 1563.682,A 0.000,B 0.000,C 90.000,E1 302.752} C_DIS
LIN {X 0.014,Y -298.362,Z 1563.667,A 0.000,B 0.000,C 90.000,E1 300.050} C_DIS
LIN {X -0.135,Y -315.853,Z 1563.654,A 0.000,B 0.000,C 90.000,E1 297.769} C_DIS
LIN {X -0.141,Y -331.051,Z 1563.643,A 0.000,B 0.000,C 90.000,E1 295.848} C_DIS
LIN {X 0.003,Y -346.215,Z 1563.633,A 0.000,B 0.000,C 90.000,E1 293.951} C_DIS
LIN {X 0.015,Y -367.018,Z 1563.620,A 0.000,B 0.000,C 90.000,E1 291.535} C_DIS
LIN {X 0.113,Y -379.999,Z 1563.612,A 0.000,B 0.000,C 90.000,E1 290.066} C_DIS
LIN {X 0.012,Y -387.478,Z 1563.607,A 0.000,B 0.000,C 90.000,E1 289.214} C_DIS
LIN {X -0.032,Y -394.453,Z 1563.602,A 0.000,B 0.000,C 90.000,E1 288.362} C_DIS
LIN {X -0.024,Y -400.786,Z 1563.597,A 0.000,B 0.000,C 90.000,E1 287.511} C_DIS
LIN {X -0.072,Y -406.359,Z 1563.593,A 0.000,B 0.000,C 90.000,E1 286.677} C_DIS
LIN {X 0.223,Y -409.653,Z 1563.589,A 0.000,B 0.000,C 90.000,E1 286.079} C_DIS
LIN {X -0.144,Y -413.816,Z 1563.585,A 0.000,B 0.000,C 90.000,E1 285.300} C_DIS
LIN {X 0.095,Y -416.156,Z 1563.582,A 0.000,B 0.000,C 90.000,E1 284.717} C_DIS
LIN {X 0.053,Y -418.192,Z 1563.579,A 0.000,B 0.000,C 90.000,E1 284.175} C_DIS
LIN {X -0.087,Y -419.823,Z 1563.576,A 0.000,B 0.000,C 90.000,E1 283.647} C_DIS
LIN {X 0.196,Y -421.025,Z 1563.573,A 0.000,B 0.000,C 90.000,E1 283.063} C_DIS
LIN {X 0.081,Y -421.819,Z 1563.570,A 0.000,B 0.000,C 90.000,E1 282.535} C_DIS
LIN {X -0.029,Y -422.100,Z 1563.567,A 0.000,B 0.000,C 90.000,E1 282.007} C_DIS
LIN {X -0.133,Y -421.901,Z 1563.564,A 0.000,B 0.000,C 90.000,E1 281.478} C_DIS
LIN {X 0.177,Y -421.219,Z 1563.561,A 0.000,B 0.000,C 90.000,E1 280.894} C_DIS
LIN {X 0.070,Y -419.879,Z 1563.558,A 0.000,B 0.000,C 90.000,E1 280.366} C_DIS
LIN {X -0.115,Y -417.970,Z 1563.555,A 0.000,B 0.000,C 90.000,E1 279.849} C_DIS
LIN {X 0.177,Y -415.394,Z 1563.552,A 0.000,B 0.000,C 90.000,E1 279.265} C_DIS
LIN {X -0.098,Y -413.864,Z 1563.550,A 0.000,B 0.000,C 90.000,E1 279.029} C_DIS
LIN {X 0.098,Y -410.170,Z 1563.547,A 0.000,B 0.000,C 90.000,E1 278.454} C_DIS
LIN {X -0.128,Y -405.654,Z 1563.544,A 0.000,B 0.000,C 90.000,E1 277.936} C_DIS
LIN {X 0.098,Y -400.358,Z 1563.541,A 0.000,B 0.000,C 90.000,E1 277.352} C_DIS
LIN {X 0.082,Y -394.462,Z 1563.538,A 0.000,B 0.000,C 90.000,E1 276.834} C_DIS
LIN {X 0.008,Y -388.427,Z 1563.535,A 0.000,B 0.000,C 90.000,E1 276.372} C_DIS
LIN {X -0.175,Y -382.218,Z 1563.533,A 0.000,B 0.000,C 90.000,E1 275.967} C_DIS
LIN {X -0.137,Y -375.880,Z 1563.531,A 0.000,B 0.000,C 90.000,E1 275.568} C_DIS
LIN {X 0.173,Y -366.096,Z 1563.528,A 0.000,B 0.000,C 90.000,E1 274.992} C_DIS
LIN {X 0.175,Y -356.271,Z 1563.525,A 0.000,B 0.000,C 90.000,E1 274.531} C_DIS
LIN {X -0.045,Y -343.489,Z 1563.522,A 0.000,B 0.000,C 90.000,E1 274.012} C_DIS
LIN {X 0.013,Y -333.681,Z 1563.520,A 0.000,B 0.000,C 90.000,E1 273.612} C_DIS
LIN {X 0.013,Y -320.624,Z 1563.518,A 0.000,B 0.000,C 90.000,E1 273.154} C_DIS
LIN {X -0.079,Y -310.415,Z 1563.516,A 0.000,B 0.000,C 90.000,E1 272.865} C_DIS
LIN {X 0.054,Y -299.725,Z 1563.514,A 0.000,B 0.000,C 90.000,E1 272.579} C_DIS
LIN {X -0.142,Y -287.832,Z 1563.513,A 0.000,B 0.000,C 90.000,E1 272.407} C_DIS
LIN {X 0.126,Y -274.506,Z 1563.512,A 0.000,B 0.000,C 90.000,E1 272.178} C_DIS
LIN {X 0.064,Y -261.397,Z 1563.512,A 0.000,B 0.000,C 90.000,E1 272.064} C_DIS
LIN {X 0.012,Y -245.714,Z 1563.511,A 0.000,B 0.000,C 90.000,E1 272.007} C_DIS
LIN {X -0.012,Y -181.261,Z 1563.511,A 0.000,B 0.000,C 90.000,E1 272.007} C_DIS
LIN {X 0.075,Y -181.567,Z 1563.503,A 0.000,B 0.000,C 90.000,E1 270.458} C_DIS
LIN {X 0.038,Y -181.175,Z 1563.490,A 0.000,B 0.000,C 90.000,E1 268.282} C_DIS
LIN {X -0.086,Y -180.842,Z 1563.472,A 0.000,B 0.000,C 90.000,E1 264.951} C_DIS
LIN {X -0.004,Y -178.951,Z 1563.444,A 0.000,B 0.000,C 90.000,E1 259.859} C_DIS
LIN {X 0.013,Y -176.856,Z 1563.425,A 0.000,B 0.000,C 90.000,E1 256.464} C_DIS
LIN {X -0.015,Y -175.518,Z 1563.411,A 0.000,B 0.000,C 90.000,E1 253.921} C_DIS
LIN {X -0.013,Y -172.255,Z 1563.387,A 0.000,B 0.000,C 90.000,E1 249.645} C_DIS
LIN {X 0.026,Y -171.734,Z 1563.382,A 0.000,B 0.000,C 90.000,E1 248.773} C_DIS
LIN {X 0.034,Y -167.330,Z 1563.353,A 0.000,B 0.000,C 90.000,E1 243.589} C_DIS
LIN {X -0.033,Y -166.715,Z 1563.349,A 0.000,B 0.000,C 90.000,E1 242.743} C_DIS
LIN {X 0.104,Y -162.695,Z 1563.324,A 0.000,B 0.000,C 90.000,E1 238.329} C_DIS
LIN {X -0.058,Y -161.386,Z 1563.314,A 0.000,B 0.000,C 90.000,E1 236.628} C_DIS
LIN {X -0.016,Y -157.379,Z 1563.290,A 0.000,B 0.000,C 90.000,E1 232.190} C_DIS
LIN {X -0.082,Y -155.372,Z 1563.275,A 0.000,B 0.000,C 90.000,E1 229.542} C_DIS
LIN {X 0.066,Y -151.712,Z 1563.250,A 0.000,B 0.000,C 90.000,E1 225.000} C_DIS
LIN {X -0.025,Y -149.903,Z 1563.235,A 0.000,B 0.000,C 90.000,E1 222.324} C_DIS
LIN {X 0.009,Y -146.762,Z 1563.210,A 0.000,B 0.000,C 90.000,E1 217.764} C_DIS
LIN {X -0.003,Y -145.329,Z 1563.195,A 0.000,B 0.000,C 90.000,E1 215.025} C_DIS
LIN {X 0.036,Y -142.411,Z 1563.164,A 0.000,B 0.000,C 90.000,E1 209.489} C_DIS
LIN {X -0.037,Y -141.395,Z 1563.148,A 0.000,B 0.000,C 90.000,E1 206.744} C_DIS
LIN {X -0.050,Y -139.354,Z 1563.112,A 0.000,B 0.000,C 90.000,E1 200.248} C_DIS
LIN {X -0.062,Y -138.794,Z 1563.097,A 0.000,B 0.000,C 90.000,E1 197.457} C_DIS
LIN {X -0.007,Y -138.346,Z 1563.055,A 0.000,B 0.000,C 90.000,E1 189.962} C_DIS
LIN {X 0.011,Y -139.378,Z 1563.009,A 0.000,B 0.000,C 90.000,E1 181.547} C_DIS
LIN {X 0.064,Y -141.269,Z 1562.972,A 0.000,B 0.000,C 90.000,E1 175.008} C_DIS
LIN {X 0.023,Y -142.635,Z 1562.957,A 0.000,B 0.000,C 90.000,E1 172.243} C_DIS
LIN {X -0.026,Y -144.964,Z 1562.931,A 0.000,B 0.000,C 90.000,E1 167.645} C_DIS
LIN {X -0.035,Y -147.591,Z 1562.911,A 0.000,B 0.000,C 90.000,E1 163.976} C_DIS
LIN {X -0.006,Y -150.208,Z 1562.891,A 0.000,B 0.000,C 90.000,E1 160.315} C_DIS
LIN {X 0.062,Y -153.593,Z 1562.870,A 0.000,B 0.000,C 90.000,E1 156.666} C_DIS
LIN {X 0.051,Y -157.009,Z 1562.851,A 0.000,B 0.000,C 90.000,E1 153.076} C_DIS
LIN {X -0.017,Y -161.128,Z 1562.831,A 0.000,B 0.000,C 90.000,E1 149.537} C_DIS
LIN {X -0.073,Y -163.229,Z 1562.821,A 0.000,B 0.000,C 90.000,E1 147.788} C_DIS
LIN {X -0.069,Y -167.661,Z 1562.801,A 0.000,B 0.000,C 90.000,E1 144.276} C_DIS
LIN {X 0.080,Y -171.484,Z 1562.787,A 0.000,B 0.000,C 90.000,E1 141.618} C_DIS
LIN {X 0.006,Y -176.414,Z 1562.768,A 0.000,B 0.000,C 90.000,E1 138.200} C_DIS
LIN {X -0.004,Y -180.708,Z 1562.754,A 0.000,B 0.000,C 90.000,E1 135.648} C_DIS
LIN {X -0.022,Y -186.113,Z 1562.735,A 0.000,B 0.000,C 90.000,E1 132.285} C_DIS
LIN {X 0.035,Y -190.750,Z 1562.721,A 0.000,B 0.000,C 90.000,E1 129.769} C_DIS
LIN {X -0.056,Y -196.504,Z 1562.703,A 0.000,B 0.000,C 90.000,E1 126.503} C_DIS
LIN {X 0.022,Y -201.280,Z 1562.689,A 0.000,B 0.000,C 90.000,E1 124.040} C_DIS
LIN {X 0.004,Y -203.699,Z 1562.682,A 0.000,B 0.000,C 90.000,E1 122.673} C_DIS
LIN {X -0.031,Y -320.132,Z 1562.682,A 0.000,B 0.000,C 90.000,E1 122.673} C_DIS
LIN {X -0.108,Y -321.110,Z 1562.681,A 0.000,B 0.000,C 90.000,E1 122.673} C_DIS
LIN {X 0.080,Y -326.353,Z 1562.680,A 0.000,B 0.000,C 90.000,E1 122.418} C_DIS
LIN {X 0.035,Y -329.447,Z 1562.679,A 0.000,B 0.000,C 90.000,E1 122.163} C_DIS
LIN {X 0.053,Y -333.127,Z 1562.676,A 0.000,B 0.000,C 90.000,E1 121.671} C_DIS
LIN {X -0.116,Y -334.781,Z 1562.674,A 0.000,B 0.000,C 90.000,E1 121.386} C_DIS
LIN {X -0.058,Y -348.950,Z 1562.655,A 0.000,B 0.000,C 90.000,E1 117.975} C_DIS
LIN {X 0.087,Y -362.036,Z 1562.640,A 0.000,B 0.000,C 90.000,E1 115.232} C_DIS
LIN {X -0.031,Y -376.667,Z 1562.625,A 0.000,B 0.000,C 90.000,E1 112.589} C_DIS
LIN {X 0.167,Y -391.069,Z 1562.613,A 0.000,B 0.000,C 90.000,E1 110.248} C_DIS
LIN {X 0.086,Y -406.888,Z 1562.600,A 0.000,B 0.000,C 90.000,E1 108.000} C_DIS
LIN {X 0.144,Y -424.235,Z 1562.588,A 0.000,B 0.000,C 90.000,E1 105.788} C_DIS
LIN {X 0.101,Y -443.230,Z 1562.576,A 0.000,B 0.000,C 90.000,E1 103.647} C_DIS
LIN {X -0.107,Y -463.240,Z 1562.565,A 0.000,B 0.000,C 90.000,E1 101.658} C_DIS
LIN {X 0.143,Y -486.385,Z 1562.553,A 0.000,B 0.000,C 90.000,E1 99.557} C_DIS
LIN {X 0.063,Y -494.069,Z 1562.550,A 0.000,B 0.000,C 90.000,E1 98.916} C_DIS
LIN {X 0.085,Y -496.000,Z 1562.548,A 0.000,B 0.000,C 90.000,E1 98.690} C_DIS
LIN {X 0.184,Y -497.473,Z 1562.547,A 0.000,B 0.000,C 90.000,E1 98.454} C_DIS
LIN {X 0.103,Y -498.689,Z 1562.546,A 0.000,B 0.000,C 90.000,E1 98.219} C_DIS
LIN {X -0.049,Y -499.572,Z 1562.544,A 0.000,B 0.000,C 90.000,E1 97.992} C_DIS
LIN {X -0.268,Y -500.489,Z 1562.542,A 0.000,B 0.000,C 90.000,E1 97.530} C_DIS
LIN {X 0.078,Y -500.395,Z 1562.539,A 0.000,B 0.000,C 90.000,E1 97.004} C_DIS
LIN {X -0.133,Y -499.278,Z 1562.536,A 0.000,B 0.000,C 90.000,E1 96.543} C_DIS
LIN {X 0.229,Y -498.283,Z 1562.535,A 0.000,B 0.000,C 90.000,E1 96.258} C_DIS
LIN {X 0.098,Y -496.934,Z 1562.534,A 0.000,B 0.000,C 90.000,E1 96.030} C_DIS
LIN {X 0.075,Y -479.236,Z 1562.519,A 0.000,B 0.000,C 90.000,E1 93.326} C_DIS
LIN {X -0.024,Y -469.393,Z 1562.510,A 0.000,B 0.000,C 90.000,E1 91.835} C_DIS
LIN {X -0.075,Y -460.806,Z 1562.503,A 0.000,B 0.000,C 90.000,E1 90.573} C_DIS
LIN {X 0.192,Y -451.802,Z 1562.496,A 0.000,B 0.000,C 90.000,E1 89.255} C_DIS
LIN {X -0.107,Y -442.427,Z 1562.489,A 0.000,B 0.000,C 90.000,E1 87.993} C_DIS
LIN {X 0.061,Y -430.709,Z 1562.480,A 0.000,B 0.000,C 90.000,E1 86.388} C_DIS
LIN {X 0.178,Y -416.988,Z 1562.469,A 0.000,B 0.000,C 90.000,E1 84.489} C_DIS
LIN {X -0.158,Y -398.094,Z 1562.454,A 0.000,B 0.000,C 90.000,E1 81.781} C_DIS
LIN {X 0.014,Y -378.605,Z 1562.437,A 0.000,B 0.000,C 90.000,E1 78.634} C_DIS
LIN {X 0.119,Y -363.600,Z 1562.422,A 0.000,B 0.000,C 90.000,E1 75.992} C_DIS
LIN {X 0.059,Y -350.708,Z 1562.409,A 0.000,B 0.000,C 90.000,E1 73.614} C_DIS
LIN {X 0.111,Y -337.974,Z 1562.396,A 0.000,B 0.000,C 90.000,E1 71.167} C_DIS
LIN {X -0.173,Y -324.246,Z 1562.380,A 0.000,B 0.000,C 90.000,E1 68.411} C_DIS
LIN {X -0.073,Y -312.707,Z 1562.366,A 0.000,B 0.000,C 90.000,E1 65.845} C_DIS
LIN {X -0.128,Y -301.244,Z 1562.351,A 0.000,B 0.000,C 90.000,E1 63.256} C_DIS
LIN {X -0.062,Y -291.381,Z 1562.338,A 0.000,B 0.000,C 90.000,E1 60.923} C_DIS
LIN {X 0.072,Y -281.519,Z 1562.325,A 0.000,B 0.000,C 90.000,E1 58.535} C_DIS
LIN {X -0.020,Y -270.561,Z 1562.310,A 0.000,B 0.000,C 90.000,E1 55.801} C_DIS
LIN {X 0.022,Y -261.166,Z 1562.296,A 0.000,B 0.000,C 90.000,E1 53.336} C_DIS
LIN {X -0.003,Y -250.711,Z 1562.280,A 0.000,B 0.000,C 90.000,E1 50.481} C_DIS
LIN {X 0.018,Y -239.686,Z 1562.262,A 0.000,B 0.000,C 90.000,E1 47.187} C_DIS
LIN {X 0.070,Y -230.646,Z 1562.246,A 0.000,B 0.000,C 90.000,E1 44.190} C_DIS
LIN {X 0.096,Y -222.360,Z 1562.229,A 0.000,B 0.000,C 90.000,E1 41.148} C_DIS
LIN {X -0.028,Y -214.838,Z 1562.212,A 0.000,B 0.000,C 90.000,E1 38.096} C_DIS
LIN {X 0.036,Y -208.122,Z 1562.194,A 0.000,B 0.000,C 90.000,E1 34.945} C_DIS
LIN {X -0.079,Y -202.198,Z 1562.177,A 0.000,B 0.000,C 90.000,E1 31.799} C_DIS
LIN {X -0.025,Y -197.023,Z 1562.159,A 0.000,B 0.000,C 90.000,E1 28.565} C_DIS
LIN {X 0.067,Y -191.562,Z 1562.136,A 0.000,B 0.000,C 90.000,E1 24.463} C_DIS
LIN {X 0.018,Y -187.075,Z 1562.113,A 0.000,B 0.000,C 90.000,E1 20.355} C_DIS
LIN {X -0.033,Y -182.713,Z 1562.085,A 0.000,B 0.000,C 90.000,E1 15.371} C_DIS
LIN {X 0.010,Y -179.344,Z 1562.057,A 0.000,B 0.000,C 90.000,E1 10.310} C_DIS
LIN {X 0.062,Y -176.566,Z 1562.024,A 0.000,B 0.000,C 90.000,E1 4.359} C_DIS
LIN {X 0.068,Y -175.533,Z 1561.974,A 0.000,B 0.000,C 90.000,E1 355.241} C_DIS
LIN {X 0.006,Y -177.711,Z 1561.931,A 0.000,B 0.000,C 90.000,E1 347.589} C_DIS
LIN {X 0.048,Y -180.822,Z 1561.903,A 0.000,B 0.000,C 90.000,E1 342.489} C_DIS
LIN {X 0.037,Y -184.593,Z 1561.879,A 0.000,B 0.000,C 90.000,E1 338.284} C_DIS
LIN {X -0.092,Y -189.238,Z 1561.856,A 0.000,B 0.000,C 90.000,E1 334.152} C_DIS
LIN {X 0.084,Y -193.706,Z 1561.838,A 0.000,B 0.000,C 90.000,E1 330.795} C_DIS
LIN {X 0.055,Y -198.798,Z 1561.820,A 0.000,B 0.000,C 90.000,E1 327.533} C_DIS
LIN {X -0.024,Y -204.684,Z 1561.802,A 0.000,B 0.000,C 90.000,E1 324.322} C_DIS
LIN {X -0.004,Y -211.314,Z 1561.784,A 0.000,B 0.000,C 90.000,E1 321.126} C_DIS
LIN {X -0.079,Y -218.859,Z 1561.767,A 0.000,B 0.000,C 90.000,E1 318.000} C_DIS
LIN {X -0.024,Y -228.246,Z 1561.747,A 0.000,B 0.000,C 90.000,E1 314.514} C_DIS
LIN {X 0.040,Y -237.600,Z 1561.730,A 0.000,B 0.000,C 90.000,E1 311.472} C_DIS
LIN {X -0.107,Y -244.171,Z 1561.720,A 0.000,B 0.000,C 90.000,E1 309.644} C_DIS
LIN {X -0.128,Y -250.207,Z 1561.712,A 0.000,B 0.000,C 90.000,E1 308.177} C_DIS
LIN {X 0.164,Y -258.759,Z 1561.702,A 0.000,B 0.000,C 90.000,E1 306.297} C_DIS
LIN {X 0.077,Y -268.418,Z 1561.692,A 0.000,B 0.000,C 90.000,E1 304.532} C_DIS
LIN {X -0.010,Y -279.169,Z 1561.682,A 0.000,B 0.000,C 90.000,E1 302.801} C_DIS
LIN {X -0.037,Y -298.168,Z 1561.667,A 0.000,B 0.000,C 90.000,E1 300.079} C_DIS
LIN {X -0.035,Y -315.667,Z 1561.654,A 0.000,B 0.000,C 90.000,E1 297.769} C_DIS
LIN {X -0.040,Y -330.899,Z 1561.644,A 0.000,B 0.000,C 90.000,E1 295.848} C_DIS
LIN {X -0.107,Y -345.792,Z 1561.633,A 0.000,B 0.000,C 90.000,E1 294.027} C_DIS
LIN {X 0.162,Y -366.491,Z 1561.620,A 0.000,B 0.000,C 90.000,E1 291.589} C_DIS
LIN {X -0.023,Y -379.430,Z 1561.612,A 0.000,B 0.000,C 90.000,E1 290.174} C_DIS
LIN {X -0.012,Y -389.247,Z 1561.606,A 0.000,B 0.000,C 90.000,E1 289.033} C_DIS
LIN {X -0.048,Y -396.109,Z 1561.601,A 0.000,B 0.000,C 90.000,E1 288.181} C_DIS
LIN {X -0.018,Y -402.279,Z 1561.596,A 0.000,B 0.000,C 90.000,E1 287.330} C_DIS
LIN {X 0.131,Y -406.013,Z 1561.593,A 0.000,B 0.000,C 90.000,E1 286.749} C_DIS
LIN {X 0.035,Y -409.385,Z 1561.590,A 0.000,B 0.000,C 90.000,E1 286.205} C_DIS
LIN {X 0.065,Y -413.674,Z 1561.585,A 0.000,B 0.000,C 90.000,E1 285.371} C_DIS
LIN {X 0.139,Y -417.175,Z 1561.581,A 0.000,B 0.000,C 90.000,E1 284.537} C_DIS
LIN {X -0.136,Y -418.195,Z 1561.579,A 0.000,B 0.000,C 90.000,E1 284.300} C_DIS
LIN {X 0.139,Y -419.914,Z 1561.576,A 0.000,B 0.000,C 90.000,E1 283.716} C_DIS
LIN {X 0.111,Y -421.241,Z 1561.573,A 0.000,B 0.000,C 90.000,E1 283.175} C_DIS
LIN {X -0.006,Y -422.123,Z 1561.570,A 0.000,B 0.000,C 90.000,E1 282.647} C_DIS
LIN {X -0.115,Y -422.527,Z 1561.567,A 0.000,B 0.000,C 90.000,E1 282.119} C_DIS
LIN {X 0.194,Y -422.456,Z 1561.564,A 0.000,B 0.000,C 90.000,E1 281.535} C_DIS
LIN {X 0.091,Y -421.863,Z 1561.561,A 0.000,B 0.000,C 90.000,E1 281.007} C_DIS
LIN {X -0.090,Y -420.705,Z 1561.558,A 0.000,B 0.000,C 90.000,E1 280.489} C_DIS
LIN {X -0.196,Y -418.934,Z 1561.555,A 0.000,B 0.000,C 90.000,E1 279.962} C_DIS
LIN {X 0.100,Y -416.515,Z 1561.552,A 0.000,B 0.000,C 90.000,E1 279.378} C_DIS
LIN {X 0.172,Y -415.062,Z 1561.551,A 0.000,B 0.000,C 90.000,E1 279.095} C_DIS
LIN {X 0.029,Y -411.557,Z 1561.548,A 0.000,B 0.000,C 90.000,E1 278.568} C_DIS
LIN {X -0.190,Y -407.123,Z 1561.545,A 0.000,B 0.000,C 90.000,E1 278.049} C_DIS
LIN {X -0.074,Y -404.746,Z 1561.543,A 0.000,B 0.000,C 90.000,E1 277.757} C_DIS
LIN {X 0.074,Y -399.071,Z 1561.540,A 0.000,B 0.000,C 90.000,E1 277.182} C_DIS
LIN {X -0.202,Y -393.170,Z 1561.537,A 0.000,B 0.000,C 90.000,E1 276.720} C_DIS
LIN {X -0.169,Y -387.141,Z 1561.535,A 0.000,B 0.000,C 90.000,E1 276.258} C_DIS
LIN {X 0.081,Y -380.785,Z 1561.532,A 0.000,B 0.000,C 90.000,E1 275.796} C_DIS
LIN {X -0.150,Y -374.329,Z 1561.530,A 0.000,B 0.000,C 90.000,E1 275.448} C_DIS
LIN {X -0.073,Y -364.668,Z 1561.527,A 0.000,B 0.000,C 90.000,E1 274.935} C_DIS
LIN {X 0.005,Y -354.844,Z 1561.525,A 0.000,B 0.000,C 90.000,E1 274.473} C_DIS
LIN {X -0.109,Y -342.270,Z 1561.522,A 0.000,B 0.000,C 90.000,E1 273.955} C_DIS
LIN {X 0.027,Y -332.605,Z 1561.520,A 0.000,B 0.000,C 90.000,E1 273.555} C_DIS
LIN {X 0.082,Y -319.467,Z 1561.517,A 0.000,B 0.000,C 90.000,E1 273.094} C_DIS
LIN {X -0.023,Y -308.943,Z 1561.516,A 0.000,B 0.000,C 90.000,E1 272.808} C_DIS
LIN {X -0.141,Y -298.190,Z 1561.514,A 0.000,B 0.000,C 90.000,E1 272.579} C_DIS
LIN {X -0.039,Y -285.567,Z 1561.513,A 0.000,B 0.000,C 90.000,E1 272.350} C_DIS
LIN {X -0.005,Y -272.140,Z 1561.512,A 0.000,B 0.000,C 90.000,E1 272.178} C_DIS
LIN {X 0.064,Y -261.462,Z 1561.512,A 0.000,B 0.000,C 90.000,E1 272.064} C_DIS
LIN {X 0.063,Y -247.959,Z 1561.511,A 0.000,B 0.000,C 90.000,E1 272.007} C_DIS
LIN {X 0.016,Y -181.260,Z 1561.511,A 0.000,B 0.000,C 90.000,E1 272.007} C_DIS
LIN {X -0.052,Y -181.581,Z 1561.501,A 0.000,B 0.000,C 90.000,E1 270.286} C_DIS
LIN {X -0.077,Y -180.897,Z 1561.473,A 0.000,B 0.000,C 90.000,E1 265.241} C_DIS
LIN {X -0.053,Y -179.847,Z 1561.459,A 0.000,B 0.000,C 90.000,E1 262.704} C_DIS
LIN {X 0.003,Y -179.030,Z 1561.445,A 0.000,B 0.000,C 90.000,E1 260.151} C_DIS
LIN {X 0.065,Y -178.679,Z 1561.441,A 0.000,B 0.000,C 90.000,E1 259.285} C_DIS
